(* CoDeSys 2.3.9.50 project: Aerosol_detection_equipment.pro *)
(* Libraries: TcFloatPC.lib 19.10.09 10:19:54, TcUtilities.lib 3.2.16 16:08:58, TcEtherCAT.lib 15.8.22 11:50:34, TcTestAndSet.lib 23.2.09 12:50:08, TcDrive.lib 25.1.17 09:42:28, TcMc2Drive.lib 9.10.17 15:27:28, TcBase.lib 14.5.09 12:14:08, TcSystem.lib 7.6.16 11:01:22, TcBaseMath.lib 27.7.04 12:07:56, TcMath.lib 23.9.04 15:15:30, TcMC2.lib 13.9.17 10:18:38, STANDARD.LIB 5.6.98 12:03:02 *)

(* Task configuration *)
TASK Standard (PRIORITY := 0, INTERVAL := T#10ms);
	MAIN
END_TASK

(* Global variable list: _01_Machine *)
VAR_GLOBAL
(*Signal*)
	stMachine						:ST_Machine;
(*Alarm*)
	arrAlarm							:ARRAY[1..MaxAlarms] OF BOOL;				(*报警号,以Excel为准*)
	arrWarning						:ARRAY[1..MaxAlarms] OF BOOL;				(*提示号,以Excel为准*)

	MSGList1 : ARRAY[1..100] OF BOOL;
	MSGList1_Alarm : BOOL;




(*Info*)
	TaskInfo						:TaskInfoCtrl;
	SysInfo							:SystemInfoCtrl;
	fPlcCycleTime_ms				:LREAL;
(* Global pulse *)
	Pulse							:PulseCtrl;		(*公共脉冲发生器*)
	nPlcTaskCycleTime_ms			:UDINT;			(*PLC周期的毫秒数*)
END_VAR

VAR_GLOBAL CONSTANT
	MaxAlarms			:UINT:=100;
END_VAR

(* Global variable list: _02_System *)
VAR_GLOBAL
	sState						:STRING(20):='MANU';		(*机台当前状态*)
	sStatus						:STRING(20):='INIT'	;			(*当前执行步骤*)

(*系统运行相关指令，面板按钮是输入来源之一*)
	bSysStart					:BOOL;		(*这个start仅指进入自动模式的启动*)
	bSysStop					:BOOL;
	bSysReset					:BOOL;
	bSysEstop					:BOOL;
	bSwitchManualMode			:BOOL;		(*打到了手动模式*)
	bSwitchAutoMode			:BOOL;		(*打到了自动模式*)
	bSysDryRunMode			:BOOL;		(*空跑模式，在触摸屏上选择，不带物料，自动运行的机械检查*)

	bSystemInAutoMode			: BOOL;		(*系统实际处于自动模式*)
	bSystemInManualMode		: BOOL;		(*系统实际处于手动模式*)
	bAutoModeRunning				:BOOL;		(*自动运行中*)

(*系统状态*)
	bGlobalErrorMark				:BOOL;		(*有报警，这个报警时会触发停机的！*)

	bSysStopFlag				:BOOL;		(*停止标记，标记出现，说明进入停机过程*)
	bStopFinished				:BOOL;		(*停止完成*)

(*指令*)
	bResetOnce					:BOOL;		(*单次复位*)
	bhasResetOnce				: BOOL;		(*已经单次复位过了*)
	bForceHomedFlag			:BOOL;		(*强制写回参信号*)
	bBuzzerSilence				:BOOL;		(*消音*)



(*自动状态*)
	eAutoStatus					:EM_Status;		(*自动模式的状态*)

(*机台状态*)
	bAllPowerOnOK				:BOOL;	(*上电检查OK*)
	bDeviceStateOK				:BOOL;	(*总线状态OK*)
	bDriveModeOK				:BOOL;	(*驱动器模式OK*)

	bAutoReady					:BOOL;		(*自动运行的位置条件OK*)
	bAllCylinderBase				:BOOL;		(*所以气缸回到初始位*)

	iSysStatus					:WORD;		(*设备状态*)
	bAirPressureOk:BOOL;(*空气压力是否到位*)



	iActPos_X_Axis					:WORD;						(*	X轴当前位置编码	*)
	iActPos_Z_Axis					:WORD;						(*	Z轴当前位置编码	*)
	iActPos_R_Axis					:WORD;						(*	R轴当前位置编码	*)
	iWarnMoveAbs							:WORD;					(*定位警告信息*)
	iAlarmNetConnect						:WORD;					(*网络连接问题报警信息*)
	iGoHomeTogether_Finish	:	WORD	;	(*一键回原点完成*)
	iGoPrepareAuto_Finish	:	WORD	;	(*一键去准备位完成*)
	iPos_X_Axis				:	WORD	;	(*模组1	X轴目标位置	*)
	iPos_Z_Axis				:	WORD	;	(*模组2	Z轴目标位置	*)
	iPos_X2_Axis				:	WORD	;	(*模组3	X轴目标位置	*)
	iPos_Y2_Axis				:	WORD	;	(*模组4	Y轴目标位置	*)
	iPos_R_Axis				:	WORD	;	(*	R轴目标位置	*)
	iX_Axis_Cmd			:	WORD	;	(*	模组1X轴目标位置运动命令	*)
	iZ_Axis_Cmd			:	WORD	;	(*	模组2Z轴目标位置运动命令	*)
	iX2_Axis_Cmd		:	WORD;		(*	模组3X轴目标位置运动命令	*)
	iY2_Axis_Cmd		:	WORD;		(*	模组4Y轴目标位置运动命令	*)
	iR_Axis_Cmd			:	WORD	;	(*	R轴目标位置运动命令	*)
	iHorizontalAxis_Cmd		:	WORD	;	(*	废物桶检测行程轴目标位置运动命令	*)
	iRotaryAxis_Cmd			:	WORD	;	(*	废物桶检测旋转轴目标位置运动命令	*)
	iLifting_PutPermit_Cmd	:	WORD	;	(*	请求吊装设备放置料筒	*)
	iLifting_GetPermit_Cmd	:	WORD	;	(*	请求吊装设备吊取料筒	*)
	iPos_CollimationAxis		:	WORD	;	(*	准直电机位置	*)
	iCollimationAxis_Cmd	:	WORD	;	(*	准直电机目标位置运动指令	*)
	iRotaryAxisRun_Cmd		:	WORD	;	(*旋转电机一直转*)
	iGoHomeTogether_Cmd	:	WORD	;	(*一键回原点*)
	iGoPrepareAuto_Cmd	:	WORD	;	(*一键去准备位*)
	iGoResetTogether_Cmd	:WORD;		(*一键复位*)
	iGoAutoTogether_Cmd		:WORD;		(*一键启动*)
	iGoStopTogether_Cmd					:WORD;		(*一键停止*)
	iAuto_Cmd				:	WORD	;	(*自动切换*)
	bGoHomeTogether_Cmd	:	BOOL	;	(*一键回原点*)
	bGoPrepareAuto_Cmd	:	BOOL	;	(*一键去准备位*)
	bAuto_Cmd				:	BOOL	;	(*自动切换*)

	bGet_Paper_Cmd:			BOOL;(*取纸*)
	bHasGot_Paper:BOOL;(*取纸完成*)

	bCollect_Cmd:BOOL;(*采集*)
	bHasCollected:BOOL;(*采集完成*)

	bPut_Paper_Cmd:			BOOL;(*放纸*)
	bHasPut_Paper:BOOL;(*放纸完成*)

	bCut_Paper_Cmd:			BOOL;(*裁纸*)
	bHasCut_Paper:BOOL;(*裁纸完成*)

	bSet_Box_Cmd:			BOOL;(*装盒子*)
	bHasSet_Box:BOOL;(*装盒子完成*)



(*报警中间变量*)
	bAxisMovingAbsAlarm			:	ARRAY[1..30] OF BOOL;

(*运行参数*)
	fSetMainVelo_Auto				: 	LREAL;			(*主轴自动速度*)
	fSetMainVelo_Manu				:	LREAL;			(*主轴手动速度*)


(**************************  工艺相关    ****************************************)

(*指令*)
	bEnaleAll						:BOOL;	(*一键使能*)
	bGoHomeTogether				:BOOL;		(*一键回原点*)
	bGoPrepareAuto					:BOOL;		(*一键初始化*)
	bGoResetTogether				:BOOL;		(*一键复位*)
	bGoAutoTogether					:BOOL;		(*一键启动*)
	bGoStopTogether					:BOOL;		(*一键停止*)
	bHeatAll							:BOOL;		(*加热所有*)

(***********************************MODBUS TCP***********************************************)

	mb_Output_Registers : ARRAY[0..255] OF WORD;
	mb_Input_Registers : ARRAY[1..255] OF WORD;

END_VAR

(* Global variable list: _03_Param *)
VAR_GLOBAL CONSTANT
	EIN                             : BOOL  := TRUE;
	AUS                             : BOOL  := FALSE;
	ANZ_SUBSSW                   : UINT   := 5;

	fCurveKp		:REAL:=6.8;		(*角度与毫米的关系*)
END_VAR

VAR_GLOBAL PERSISTENT
	iAxisSoftLimitSwitch_Neg	:ARRAY[1..5] OF BOOL;	(*软限位正限开关*)
	iAxisSoftLimitSwitch_Pos	:ARRAY[1..5] OF BOOL;	(*软限位负限开关*)

	iAxisSoftLimitSwitch_Neg1	:ARRAY[1..5] OF WORD;	(*软限位正限开关*)
	iAxisSoftLimitSwitch_Pos1	:ARRAY[1..5] OF WORD;	(*软限位负限开关*)
	fSaveBias	:ARRAY[1..5] OF REAL;
END_VAR

VAR_GLOBAL

(*运行时数据状态*)
	iAxisSoftLimitSwitch_Neg_Old	:ARRAY[1..5] OF BOOL;	(*软限位正限开关*)
	iAxisSoftLimitSwitch_Pos_Old	:ARRAY[1..5] OF BOOL;	(*软限位负限开关*)
	iMacStateForHmi				:WORD;(*机器状态给HMI*)
END_VAR

(* Global variable list: _04_Motion *)
VAR_GLOBAL
	AxisArr					:ARRAY[1..MaxAxes] OF  axis_ref;		(*PTP轴*)
	Axis_Interface			: ARRAY [1..MAXAxes] OF ST_Axis;		(*轴的PTP控制接口*)
(*功能块定义*)
	aMC_Power				:ARRAY[1..MaxAxes] OF MC_Power;
	aMC_Jog				:ARRAY[1..MaxAxes] OF MC_Jog;
	aMC_Reset				:ARRAY[1..MaxAxes] OF MC_Reset;
	aMC_Halt				:ARRAY[1..MaxAxes] OF MC_Halt;
	aMC_Stop				:ARRAY[1..MaxAxes] OF MC_Stop;
	aMC_SetPos				:ARRAY[1..MaxAxes] OF MC_SetPosition;
	aMC_MoveAbsolute		:ARRAY[1..MaxAxes] OF MC_MoveAbsolute;
	aMC_MoveRelative		:ARRAY[1..MaxAxes] OF MC_MoveRelative;
	aMC_MoveVelocity		:ARRAY[1..MaxAxes] OF MC_MoveVelocity;
	aMC_SetHomeFlag		:ARRAY[1..MaxAxes] OF MC_Home;
	aMC_Home				:ARRAY[1..MaxAxes] OF MC_Home;
	aMC_GearInDyn			:ARRAY[1..MaxAxes] OF MC_GearInDyn;			(*电子齿轮轮耦合*)
	aMC_GearOut			: ARRAY[1..MaxAxes] OF MC_GearOut;		(*电子齿轮轮解耦合*)
	aMC_SoeReset			:ARRAY[1..MaxAxes] OF FB_SoEReset;		(*倍福驱动器复位*)

(*公共状态参数*)
 	Axis_Has_error		:BOOL;		(*任何一根轴有任何错误*)
	Axis_Homing			:BOOL;		(*任何一根轴在回参*)
	All_Enable_OK		:BOOL;		(*所有轴使能成功*)
	All_Homed_OK		:BOOL;		(*所有轴回零成功*)
	bAllAxisAtZero		:BOOL;		(*所有轴都在0位*)
	AllAxesStandStill		:BOOL;		(*所有轴静止*)
(*公共CMD参数*)
	bEnableAll	:	BOOL;	(*使能所有轴*)
(*气缸*)
	stCtrlCylinder	:ARRAY[1..NumOfCylinders]OF ST_Cylinder_Ctrl;
	fbCylinder		:ARRAY[1..NumOfCylinders]OF FB_Cylinder;
END_VAR

VAR_GLOBAL CONSTANT
	MaxAxes							:UINT:=5;		(*轴数，不同于驱动器数，后者是物理轴的个数*)
	NumOfDrives							:UINT:=5;		(*实际驱动器数*)
	MinHomeAxis	:UINT:=1;		(*最小回原点轴*)
	MaxHomeAxis	:UINT:=8;		(*最大回原点轴*)
	NumOfCylinders						:UINT:=38;		(*气缸数*)
END_VAR

(* Global variable list: _05_IO *)
VAR_GLOBAL
	(*数字量输入*)
	El1889s			AT %I*		:ARRAY[1..NumOfDiModule,1..NumOfChannel]OF BOOL;
	(*数字量输出*)
	El2889s 			AT%Q*		:ARRAY[1..NumOfDoModule,1..NumOfChannel]OF BOOL;
	(*模拟量输入*)
	El3064			AT %I*		:ARRAY[1..4]OF INT;
	(*实际驱动器作为EtherCAT伺服的个数  ETHERCAT状态*)
	DrivesOP 		AT %I*		:ARRAY[1..NumOfDrives]OF UINT;
	(*驱动器的模式输出，8为位置模式*)
	iSetDriveMode 	AT %Q*		:ARRAY [1..NumOfDrives] OF SINT := NumOfDrives(CSP);
	(*驱动器返回的控制模式*)
	iActDriveMode	AT%I*		:ARRAY[1..NumOfDrives]OF SINT;
	(*驱动器上的IO监控，EL2521不包含*)
	iDriveDI			AT%I*  :ARRAY [1..NumOfDrives] OF INT;
	(*驱动器上的电流监控，EL2521不包含*)
	iMotorTorque		 AT%I*  :ARRAY [1..NumOfDrives] OF INT;

END_VAR


VAR_GLOBAL CONSTANT
	NumOfDiModule		:UINT:=7;		(*DI输入模块总数*)
	NumOfDoModule		:UINT:=3;		(*DO输出模块总数*)
	NumOfAiModule		:UINT:=0;		(*DI输入模块总数*)
	NumOfChannel		:UINT:=16;		(*IO模块的通道数*)

	iEcatOp				:UINT:=8;
	CSP					:USINT:=8;
	CSV					:USINT:=9;
	CST					:USINT:=10;
END_VAR

(* Global variable list: _06_Hmi *)
VAR_GLOBAL
(***********************HMI变量****************************)
(********  指令 ***********)
	stHmiCmd			:	ST_HmiCmd;
	stHmiAxisCmd			:	ARRAY[1..MaxAxes] OF ST_AxisCmd;
(********  显示 ***********)
	stHmiDisplay				:	ST_HmiDisplay;
	stAxisDisplay			:	ARRAY[1..MaxAxes] OF ST_AxisDisplay;
END_VAR


VAR_GLOBAL PERSISTENT
(********  参数 ***********)
	stAxisParam			:	ARRAY[1..MaxAxes] OF ST_AxisParam;
END_VAR

(* Global variable list: TwinCAT_Configuration *)
(* Generated automatically by TwinCAT - (read only) *)
VAR_CONFIG
	.AxisArr[1].PlcToNc AT %QB53 : PLCTONC_AXIS_REF;	(*  ~ {LinkedWith:TINC^NC-Task 1 SAF^Axes^Axis 1^Inputs^Axis 1_FromPlc} *)
	.AxisArr[1].NcToPlc AT %IB155 : NCTOPLC_AXIS_REF;	(*  ~ {LinkedWith:TINC^NC-Task 1 SAF^Axes^Axis 1^Outputs^Axis 1_ToPlc} *)
	.AxisArr[2].PlcToNc AT %QB181 : PLCTONC_AXIS_REF;	(*  ~ {LinkedWith:TINC^NC-Task 1 SAF^Axes^Axis 2^Inputs^Axis 2_FromPlc} *)
	.AxisArr[2].NcToPlc AT %IB283 : NCTOPLC_AXIS_REF;	(*  ~ {LinkedWith:TINC^NC-Task 1 SAF^Axes^Axis 2^Outputs^Axis 2_ToPlc} *)
	.AxisArr[3].PlcToNc AT %QB309 : PLCTONC_AXIS_REF;	(*  ~ {LinkedWith:TINC^NC-Task 1 SAF^Axes^Axis 3^Inputs^Axis 3_FromPlc} *)
	.AxisArr[3].NcToPlc AT %IB411 : NCTOPLC_AXIS_REF;	(*  ~ {LinkedWith:TINC^NC-Task 1 SAF^Axes^Axis 3^Outputs^Axis 3_ToPlc} *)
	.AxisArr[4].PlcToNc AT %QB437 : PLCTONC_AXIS_REF;	(*  ~ {LinkedWith:TINC^NC-Task 1 SAF^Axes^Axis 4^Inputs^Axis 4_FromPlc} *)
	.AxisArr[4].NcToPlc AT %IB539 : NCTOPLC_AXIS_REF;	(*  ~ {LinkedWith:TINC^NC-Task 1 SAF^Axes^Axis 4^Outputs^Axis 4_ToPlc} *)
	.AxisArr[5].PlcToNc AT %QB565 : PLCTONC_AXIS_REF;	(*  ~ {LinkedWith:TINC^NC-Task 1 SAF^Axes^Axis 5^Inputs^Axis 5_FromPlc} *)
	.AxisArr[5].NcToPlc AT %IB667 : NCTOPLC_AXIS_REF;	(*  ~ {LinkedWith:TINC^NC-Task 1 SAF^Axes^Axis 5^Outputs^Axis 5_ToPlc} *)
	.El1889s AT %IB0 : ARRAY [1..7, 1..16] OF BOOL;
	.El2889s AT %QB0 : ARRAY [1..3, 1..16] OF BOOL;
	.El3064 AT %IB112 : ARRAY [1..4] OF INT;
	.DrivesOP AT %IB120 : ARRAY [1..5] OF UINT;
	.iSetDriveMode AT %QB48 : ARRAY [1..5] OF SINT;
	.iActDriveMode AT %IB130 : ARRAY [1..5] OF SINT;
	.iDriveDI AT %IB135 : ARRAY [1..5] OF INT;
	.iMotorTorque AT %IB145 : ARRAY [1..5] OF INT;
END_VAR

(* Data type in 01_States *)
TYPE EM_State :	(*机台或者部件的几种状态*)
(
	PowerOn,
	ConnectionTest,
	Init,
	Manu,
	Auto,
	Error
);
END_TYPE

(* Data type in 01_States *)
TYPE EM_Status :	(*自动模式下的几个流程*)
(
	AUTO_STOP       :=   0,
	AUTO_W_RUN      :=   2,
	AUTO_RUN        :=   3,
	AUTO_W_HALT     :=   4,
	AUTO_HALT       :=   5,
	AUTO_W_STOP     :=   6
);
END_TYPE

(* Data type in 04_AxisControl *)
TYPE ST_Axis :	(*Johnson made this on 2017-01-17*)
STRUCT
(*status*)
	AxisName		:STRING(31);		(*轴名称*)
	AxisID			:UDINT;		(*轴在NC中的编号*)

	Axis_Limit_Neg	:BOOL;		(*负限位触发信号*)
	Axis_Limit_Pos	:BOOL;		(*正限位触发信号*)
	Axis_HomeSwitch	:BOOL;		(*原点触发信号*)
	Axis_Ready		:BOOL;
	Axis_Err			:BOOL;
	Axis_ErrID		:UDINT;

	Axis_Homed		:BOOL;
	Axis_Homing		:BOOL;
	Axis_Coupled		:BOOL;
	Axis_NotMoving	:BOOL;

	fActPos			:LREAL;
	fActPosModbus			:WORD;
	fActVelo			:LREAL;
	fScaleFactor		:LREAL;
(*Command*)
	bEnable			:BOOL;		(*使能*)
	bEnableFw		:BOOL:=TRUE;		(*正向使能*)
	bEnableBw		:BOOL:=TRUE;		(*负向使能*)
	bJog_Fw			:BOOL;		(*正向点动*)
	bJog_Bw		:BOOL;		(*反向点动*)

	bHalt			:BOOL;	(*暂停*)
	bStop			:BOOL;	(*停止*)
	bReset			:BOOL;	(*复位*)

	bMoveAbs		:BOOL;	(*运行绝对位置*)
	bMoveRel		:BOOL;	(*运行当对位置*)
	bMoveVelo		:BOOL;	(*向一个方向持续运行，方向由前面的正向点动或者反向点动设置*)

	bHome			:BOOL;		(*启动回参*)
	bSetPos			:BOOL;		(*设置轴当前的位置为一个绝对位置*)

	bCamIn			:BOOL;
	bCamOut		:BOOL;

	bGearIn			:BOOL:=FALSE;
	bGearOut		:BOOL:=FALSE;

	fGearInDynAcc	:LREAL:=50000;
	fGearInDynDec	:LREAL:=50000;
	fGearRatio		:LREAL;		(*电子齿轮耦合齿轮比*)

	nCmdMode		:SINT;(*8=CSP位置, 9=CSV,10=CST力矩*)
(*Parameter*)
	fOverride			 :LREAL:=100;		(*MC_power中实际倍率的设定，默认值为100*)
	fPositon_of_Abs	 :LREAL;		(*绝对位置位移*)
	fPosition_of_Rel	 :LREAL;		(*相对位置位移*)
	fVelocity_of_Abs	 :LREAL:=5;		(*位置移动速度，包含相对位移和绝对位移指令的速度*)
	fVelocity_of_Rel	 :LREAL;		(*位置移动速度，包含相对位移和绝对位移指令的速度*)
	fVelocity_of_Velo	 :LREAL;		(*速度指令下的运动速度，用在mc_movevelocity里面*)
	fVelocity_of_Jog	 :LREAL:=5;		(*手动点动速度，可以在程序里面设置不同值*)

	fAcc				:LREAL:=0;(*0代表使用SystemManager里面的参数*)
	fDec			:LREAL:=0;
	fJerk			:LREAL:=0;
	fPosition_ToBeSet	:LREAL;		(*setpos功能块将轴当前的位置设置为这个变量*)
	fRefPos				:LREAL:=0;		(*使用TwinCAT PLC的MC_Home回零时，将外部信号设成这个值*)

	bInVelo			:BOOL;		(*速度模式，达到了速度*)
END_STRUCT
END_TYPE

(* Data type in 05_Function/02_Axis *)
TYPE ST_AxisCmd :
STRUCT
(*Command*)
	bEnable				:BOOL(*:=TRUE*);
	bJog_Fw			:BOOL;		(*正向点动*)
	bJog_Bw			:BOOL;		(*反向点动*)
	bJog_InchingFw			:BOOL;		(*正向寸动*)
	bJog_InchingBw			:BOOL;		(*反向寸动*)
	bMoveToZero				:BOOL;		(*回原点*)		(*正负极直线电机回原点，纠偏和切刀回原点，短路测试电机回原点，叠台...*)
	bMoveAbs				:BOOL;
	bMoveRel				:BOOL;
	bReset					:BOOL;
	bHome					:BOOL;
	bSetPos					:BOOL;
	bSetBiasBnt			:BOOL;		(*保存原点按钮*)
END_STRUCT
END_TYPE

(* Data type in 05_Function/02_Axis *)
TYPE ST_AxisDisplay :
STRUCT
(*DisPlay*)
	bError			:BOOL;		(*报错*)
	bEnabled		:BOOL;		(*使能*)
	bHoming			:BOOL;		(*回参中*)
	bHomed			:BOOL;		(*回参完成*)
	bMoiving		:BOOL;		(*移动中*)
	bPosLimit		:BOOL;
	bNegLimit		:BOOL;
	udiErrorId		:UDINT;		(*轴错误代码*)

	fActPos	 		:REAL:=15;			(*轴当前位置*)
(*	fActModPos		:REAL:=0;	*)
	fActVelo		:REAL:=5;			(*轴当前速度*)
	fOverride		:REAL:=100;			(*轴当前速比值*)

END_STRUCT
END_TYPE

(* Data type in 05_Function/02_Axis *)
TYPE ST_AxisParam :
STRUCT
(*Parameter，头两个参数可以用触摸屏上设置*)
	fVelocity_of_Jog	 		:LREAL:=4;			(*手动点动速度，可以在程序里面设置不同值*)
	fInchingDistance			:LREAL:=1;			(*寸动距离，可以在程序里面设置不同值*)
	fVelo_of_Posi			:REAL:=15;		(*手动定位速度*)

	fVelo_of_Auto		:LREAL:=6;		(*自动速度*)
	fVelocity_of_Abs		:LREAL:=6;
	fTargetPos				:LREAL;

	fOverride				:LREAL:=100;			(*实际倍率的设定，默认值为100*)
	SavedPosition			:LREAL:=0;
	iTargetNr				:UINT;
	ZeroPos				:REAL;		(*零位，原点开关决定*)
	StandbyPos			:REAL;		(*待机位*)
	WorkPos1			:REAL;		(*工位1*)
	WorkPos2			:REAL;		(*工位2*)
	WorkPos3			:REAL;		(*工位3*)

	fTargetPosi			:REAL;		(*目标定位*)
END_STRUCT
END_TYPE

(* Data type in 04_AxisControl *)
TYPE ST_Cylinder_Ctrl :	(*Johnson made this on 2017-01-17*)
STRUCT
(*From DI*)
	DiBaseLimit				:BOOL;		(*负限位触发信号*)
	DiWorkLimit				:BOOL;		(*正限位触发信号*)

(*To Do*)
	DoAct			:BOOL;		(*动作*)
	DoBack			:BOOL;		(*回到base位*)

(*To PLC status*)
	CylinderName		:STRING(31);		(*气缸名称*)
	CylinderID			:UDINT;				(*气缸编号*)

	Cylinder_Limit_Base	:BOOL;		(*负限位触发信号*)
	Cylinder_Limit_Work	:BOOL;		(*正限位触发信号*)
	CylinderAlarm_TimeOut	:BOOL;			(*气缸动作超时*)

(*PLC commmand*)
	bAct			:BOOL;		(*动作*)
	bBack			:BOOL;		(*回到base位*)
	bSwitch			:BOOL;		(*切换*)


(*Parameter*)
	bContinue				:BOOL;	(*是否连续运动气缸*)
	fTimeOfContinue			:REAL:=1;
	fTimeOfOvertime			:REAL:=1;		(*单位秒*)

END_STRUCT
END_TYPE

(* Data type in 05_Function/01_Machine *)
TYPE ST_HmiCmd :
STRUCT

(***************************************************   系统    ********************************************)

	bStart		:BOOL;
	bStop		:BOOL;
	bReset		: BOOL;		(*HMI上的复位*)
	bEstop		: BOOL;		(*HMI上的急停*)
	bNtReboot		: BOOL;		(*系统重启*)
	bNtShutdown	: BOOL;		(*系统关机*)
	bSaveData		: BOOL;		(*保存系统设置参数*)
	bSilence			: BOOL;		(*消音按钮*)
END_STRUCT
END_TYPE

(* Data type in 05_Function/01_Machine *)
TYPE ST_HmiDisplay :
STRUCT

(***************************************************  设备状态     ********************************************)

	bAll_Enable_OK				:BOOL;	(*所有轴使能成功*)
	bAll_Homed_OK				:BOOL;	(*所有轴回零成功*)
	bAutoReady					:BOOL;	(*运行准备信号，满足了打到自动的准备条件*)
	bAutoSwitch				:BOOL;	(*在界面上显示当前旋转开关处于手动还是自动,True为自动，false为手动*)
	bAutoMode					:BOOL;	(*设备进入了自动模式*)
	bAutoRunning  				:BOOL;	(*自动运行中*)
	bHeartBeat					:BOOL;
	iMachineState			:		UINT;		(*机台状态*)
(***************************************************  系统     ********************************************)
	sProgram_Vision				:STRING;	(*程序版本号*)


END_STRUCT
END_TYPE

(* Data type in 03_Machine *)
TYPE ST_Machine :
STRUCT

(***************************************************   DI    ********************************************)
	btnStart			:BOOL;	(*	启动按钮	*)
	btnStop			:BOOL;	(*	停止按钮	*)
	btnReset		:BOOL;	(*	复位按钮	*)
	bswAutoSwitch	:BOOL;	(*	手自动切换按钮	*)
	btnEstop		:BOOL;	(*	急停按钮	*)
	bSingle			:BOOL;



(***************************************************   DO    ********************************************)

	boLamp_Red		:BOOL;	(*	灯柱-红	*)
	boLamp_Green	:BOOL;	(*	灯柱-绿	*)
	boLamp_Yellow	:BOOL;	(*	灯柱-黄	*)
	boBuzzer		:BOOL;	(*	蜂鸣器	*)
	boBtnStartLed	:BOOL;	(*启动按钮指示灯，绿色*)
	boBtnStopLed	:BOOL;	(*停止按钮指示灯，红色*)
	boBtnResetLed	:BOOL;	(*复位按钮指示灯，橙色*)
END_STRUCT
END_TYPE

(* POU MAIN, ST *)
PROGRAM MAIN
VAR
	MainState					:EM_State;	(*主程序步，其他程序可以读*)
	bFirstCycle: BOOL:=TRUE;	(*初始化用的*)
(*保存掉电保持参数*)
	FB_WritePersistentData1: FB_WritePersistentData;
	tCycleTimer:TON;
	bWrite: BOOL;

(*系统重启*)
	tNtDelayReset:TON;
	bReboot: BOOL;	(*重启系统的变量*)
	NT_Reboot1: NT_Reboot;

(*系统关机*)
	NT_Shutdown1: NT_Shutdown;
	tNtDelayShutdown: TON;
	bShutdown: BOOL;

(*远程桌面接管*)
	OpenRemoteDesktop: NT_StartProcess;
	timerHMI	:TON;

(*设置系统时间*)
	TimeToBeSet: TIMESTRUCT;
	bSetTime: BOOL;
	NT_SetLocalTime_1: NT_SetLocalTime;
(*系统时间获取*)
	NT_GetTime1: NT_GetTime;
	GetTimeStartDelay:TON;
	TIMESTR1				:TIMESTRUCT;

	i: UINT;

(*
(*计算加工时间相关变量*)
	j:UINT;(*表格的FOR序号*)
	n:UINT:=1;
	rtrigAutoRunning:R_TRIG;	(*自动运行上升沿*)
	ftrigAutoRunning:F_TRIG;	(*自动运行下升沿*)
	nStopLock: BOOL;
	itets: UINT;
(*其它*)
	R_TRIG_Enabled: R_TRIG;
	BalanceLumpDeclineDelay:TON;(*配重块下降到下限传感器位置后延时一定时间才停止*)
	nParameterUpdateTop:BOOL;(*参数被更改，提醒用户更新运行数据*)
	ActTableModeNumber: BOOL;	(*表格序号至少一个被激活*)
*)
	rtrigStart,rtrigReset,rtrigStop: R_TRIG;
	fTrigAutoManulMode: F_TRIG;
	rTrigAutoManualMode: R_TRIG;
	tDelayManualMode:TON;(*打到手动的延时*)
(*Lamp and Buzzer*)
	eStepBuzze: UINT;
	rTrigBuzze: R_TRIG;
	tDelayBuzze: TON;



	LagDistance_ZM: LREAL;
	LagDistance_CM: LREAL;
	FirstCycle_Step: UINT;
	R_TRIGbDriveModeOK:R_TRIG;
	tDelay:TON;
END_VAR
PRG_IO.Input();
PRG_Alarm();
PRG_Monitor();
PRG_Auto.Act_Modbus_TCP();
MAIN._NT;
MAIN.Command;
MAIN.Status;

CASE MainState OF
PowerOn:
	PRG_Power();
	MainState:=ConnectionTest;

ConnectionTest:
	IF bDeviceStateOK AND bDriveModeOK  THEN
		bResetOnce:=TRUE;
		MainState:=INIT;
		PRG_ServOn();
	END_IF

INIT:	(*程序的初始化处理，并非机器的工艺初始化*)
	PRG_Init();
	IF All_Enable_OK OR bHasResetOnce   THEN
		MainState:=MANU;
	ELSIF Axis_Has_error THEN
		MainState:=ConnectionTest;		(*轴有错就再复位一次,这个时针对有的驱动在PLC之前启动好，PLC连接时会报通讯错误，需要复位一次*)
		bHasResetOnce:=TRUE;
	END_IF

MANU:
(*手动模式*)
	PRG_Manual;
	IF bSysEstop  THEN			(*急停也是从手动中进入的*)
		MainState:=ERROR;
	ELSIF
		bSwitchAutoMode
		AND NOT bGlobalErrorMark
		AND NOT bSysEstop
		AND bAutoReady
	THEN
		MainState:=AUTO;
	END_IF

AUTO:
	PRG_Auto();
	IF  bSysEstop (*AND bStopFinished*) THEN	(*急停触发，并且停好了*)
		MainState:=ERROR;
	ELSIF bSwitchManualMode AND NOT bStopFinished THEN
		MainState:=MANU;
	END_IF
ERROR:
	PRG_Estop();
	IF NOT bSysEstop THEN
		MainState:=PowerOn;
		bResetOnce:=TRUE;
	END_IF
END_CASE


IF( bSysEstop AND MainState<>AUTO) (*OR bGlobalErrorMark *)THEN		(*非自动模式下的急停处理*)
	MainState:=ERROR;
END_IF
PRG_M_Function();
PRG_PTP();
PRG_Auto.Act_Run();
PRG_IO.Output();
END_PROGRAM
ACTION _NT:
(*系统重启，CE远程桌面，系统时间，定时保存掉电数据，等系统常规动作*)

tNtDelayReset(IN:=bReboot , PT:=t#3s , Q=> , ET=> );
NT_Reboot1(
	NETID:='' ,
	DELAY:= ,
	START:=(*tNtDelayReset.Q  ,*),
	TMOUT:=DEFAULT_ADS_TIMEOUT ,
	BUSY=> ,
	ERR=> ,
	ERRID=> );

tNtDelayShutdown(IN:=bShutdown , PT:=t#0.5s , Q=> , ET=> );
NT_Shutdown1(
	NETID:= ,
	DELAY:= ,
	START:=tNtDelayShutdown.Q,			(*针对win7系统用的，CE系统直接断电*)
	TMOUT:=DEFAULT_ADS_TIMEOUT ,
	BUSY=> ,
	ERR=> ,
	ERRID=> );

(******************* 开启CE系统远程桌面  ******************************************)
timerHMI(IN:=bFirstCycle, PT:=T#2S);
(*IF timerHMI.Q THEN
	bFirstCycle:=FALSE;
END_IF*)
OpenRemoteDesktop(
	NETID:='' ,
	PATHSTR:='\windows\CerDisp.exe' ,
	DIRNAME:='\windows' ,
	COMNDLINE:= ,
	START:=(*timerHMI.Q*) ,		(*建议第一次通过程序手动开启远程桌面之后，再修改注册表种launch90的值，以及增加Enable远程的注册表文件到regfile中来实现*)
	TMOUT:= ,
	BUSY=> ,
	ERR=> ,
	ERRID=> );
(********************** 获取系统时间   ***************************************)


GetTimeStartDelay(IN:=NOT GetTimeStartDelay.Q  , PT:=T#2s , Q=> , ET=> );
NT_GetTime1(
	NETID:= ,
	START:=GetTimeStartDelay.Q ,
	TMOUT:= , 
	BUSY=> ,
	ERR=> ,
	ERRID=> ,
	TIMESTR=>TIMESTR1 );

TIMESTR1.wYear;		(*年*)
TIMESTR1.wMonth;		(*月*)
TIMESTR1.wDay;		(*日*)
TIMESTR1.wHour;		(*时*)
TIMESTR1.wMinute;		(*分*)
TIMESTR1.wSecond;		(*秒*)
TIMESTR1.wMilliseconds;	(*毫秒*)
TIMESTR1.wDayOfWeek;	(*星期*)

(********************** 设置系统时间   ***************************************)
NT_SetLocalTime_1(
	NETID:= , 
	TIMESTR:=TimeToBeSet ,
	START:=bSetTime ,
	TMOUT:=t#500ms ,
	BUSY=> , 
	ERR=> ,
	ERRID=> );
TimeToBeSet.wYear;			(*年*)
TimeToBeSet.wMonth;		(*月*)
TimeToBeSet.wDay;			(*日*)
TimeToBeSet.wHour;			(*时*)
TimeToBeSet.wMinute;		(*分*)
TimeToBeSet.wSecond;		(*秒*)
TimeToBeSet.wMilliseconds;	(*毫秒*)
TimeToBeSet.wDayOfWeek;	(*星期*)

(***********************  保存掉电保持数据   **************************************)
tCycleTimer(IN:=NOT tCycleTimer.Q , PT:=t#60s , Q=>bWrite , ET=> );
FB_WritePersistentData1(
	NETID:='' ,
	PORT:=801 ,
	START:=bWrite OR stHmiCmd.bSaveData OR SystemtaskInfoArr[1].firstCycle  ,
	TMOUT:=t#500ms ,
	MODE:=SPDM_2PASS ,
	BUSY=> ,
	ERR=> ,
	ERRID=> );
(**********************  系统周期时间获取   ***************************************)
nPlcTaskCycleTime_ms:=SystemtaskInfoArr[1].cycleTime/10000;


(******************* 伺服位置设置********************)
R_TRIGbDriveModeOK(CLK:=(bDriveModeOK), Q=> );
IF (R_TRIGbDriveModeOK.Q AND timerHMI.Q) OR (FirstCycle_Step=0 AND MainState=MANU)  THEN
		FirstCycle_Step:=100;
END_IF



tDelay(IN:= , PT:=t#20ms , Q=> , ET=> );

CASE FirstCycle_Step OF
0:
;
100:
	tDelay.IN:=TRUE;
	IF tDelay.Q THEN
		FirstCycle_Step:=110;
	END_IF
110:
	tDelay.IN:=FALSE;
	FOR i:=1 TO 5 DO
		Axis_Interface[i].fPosition_ToBeSet := -fSaveBias[i]+AxisArr[i].NcToPlc.ActPos;
	END_FOR
	FirstCycle_Step:=200;
200:
	FOR i:=1 TO 5 DO
		Axis_Interface[i].bSetPos:=TRUE;(*触发信号*);
	END_FOR
	FirstCycle_Step:=300;
300:
	bFirstCycle:=FALSE;
	FirstCycle_Step:=400;
400:
	;
END_CASE
END_ACTION
ACTION Command:
(*系统状态切换按钮的响应与信号汇总，以及指示灯的输出*)

rtrigStart(CLK:=stMachine.	btnStart OR stHmiCmd.bStart , Q=> );		(*如果有其他HMI触发的信号也写到此处*)
rtrigStop(CLK:=stMachine.	btnStop OR stHmiCmd.bStop, Q=> );
rtrigReset(CLK:=stMachine.	btnReset OR stHmiCmd.bReset OR bResetOnce, Q=> );

tDelayManualMode(IN:=NOT (stMachine.bswAutoSwitch OR bAuto_Cmd),PT:=t#1s,Q=>,ET=>);(*下降沿延迟*)
rTrigAutoManualMode(CLK:=stMachine.bswAutoSwitch OR bAuto_Cmd, Q=> );		(*打到自动的上升沿*)
fTrigAutoManulMode(CLK:=tDelayManualMode.Q, Q=> );		(*下降沿信号*)


IF bResetOnce THEN
	bResetOnce:=FALSE;		(*触发后将信号复位掉*)
END_IF

(*模式选择*)
IF  rTrigAutoManualMode.Q THEN
	bSwitchAutoMode:=TRUE;
	bSwitchManualMode:=FALSE;
ELSIF tDelayManualMode.Q AND NOT stMachine.bswAutoSwitch  THEN
	bSwitchAutoMode:=FALSE;
	bSwitchManualMode:=TRUE;
END_IF

(*自动运行判定*)
bAutoModeRunning;
bSystemInManualMode:=(MainState=MANU);
bSystemInAutoMode:=(MainState=AUTO);


(*单次触发的信号*)
bSysStart:=rtrigStart.Q ;
bSysStop:=rtrigStop.Q;
bSysReset:=rtrigReset.Q ;
bSysEstop:=stMachine.btnEstop;




bBuzzerSilence:=stHmiCmd.bSilence;	(*触摸屏选择消音,彻底不报警*)




(********************************** Systemfunctions **********************************************************)
	SysInfo(
		Reset				:= ,
		TimeStampTrig		:= Pulse._100ms.RT,
		RunTimeNo			=> ,
		ProjectName			=> ,
		NumberOfTasks		=> ,
		OnlineChangeCount	=> ,
		RetainVarErr		=> ,
		PersistenVarErr		=> ,
		TimeStampDT			=> ,
		TimeStamp			=> ,
		TimeStr				=> ,
		DateStr				=> ,
		TimeStamp2			=> ,
		TimeStruct			=> ,
		MonthDays			=> ,
		LeapYear			=> ,
		WeekOfYear			=> ,
		timezoneId			=>);

	TaskInfo(
		index				=> ,
		active				=> ,
		taskName			=> ,
		firstCycle			=> ,
		cycleTimeExceeded	=> ,
		cycleTime			=> ,
		lastExecTime		=> ,
		priority			=> ,
		cycleCount			=> );

	Pulse(
		BlinkSlow			=> ,
		Blink				=> ,
		BlinkFast			=> );
END_ACTION
ACTION Status:
(*系统灯*)

CASE eStepBuzze OF
	0:
	(*系统故障或者急停时*)
		rTrigBuzze(CLK:=bGlobalErrorMark OR bSysEstop  , Q=> );
		IF rTrigBuzze.Q
		THEN
			eStepBuzze:=10;
			tDelayBuzze(IN:= TRUE, PT:=t#3s , Q=> , ET=> );
		END_IF
	10:
		stMachine.boBuzzer:=bGlobalErrorMark AND Pulse._1s.Q;
		tDelayBuzze(IN:= TRUE, PT:=t#3s , Q=> , ET=> );
		IF tDelayBuzze.Q
		THEN
			eStepBuzze:=0;
			tDelayBuzze(IN:= FALSE, PT:=t#3s , Q=> , ET=> );
			stMachine.boBuzzer:=FALSE;
		END_IF
END_CASE


IF bGlobalErrorMark
THEN										(*报错，红灯*)
	stMachine.boLamp_Green:=FALSE;
	stMachine.boLamp_Red:=TRUE;
	stMachine.boLamp_Yellow:=FALSE;

	stMachine.boBtnStopLed:=TRUE;
	stMachine.boBtnStartLed:=FALSE;
	stMachine.boBtnResetLed:=FALSE;
ELSIF MainState=AUTO (*AND bAutoModeRunning*)					(*自动模式，并且运动起来了*)
THEN
	stMachine.boLamp_Green:=bAutoModeRunning;
	stMachine.boLamp_Red:=FALSE;
	stMachine.boLamp_Yellow:=FALSE;

	stMachine.boBtnStopLed:=FALSE;
	stMachine.boBtnStartLed:=TRUE;
	stMachine.boBtnResetLed:=FALSE;
ELSE										(*手动，黄灯*)
	stMachine.boLamp_Green:=FALSE;
	stMachine.boLamp_Red:=FALSE;
	stMachine.boLamp_Yellow:=TRUE;

	stMachine.boBtnStopLed:=FALSE;
	stMachine.boBtnStartLed:=FALSE;
	stMachine.boBtnResetLed:=TRUE;
END_IF


CASE MainState OF
PowerOn:			stHmiDisplay.iMachineState:=0;
ConnectionTest:		stHmiDisplay.iMachineState:=1;
MANU:			stHmiDisplay.iMachineState:=2;iSysStatus:=1;
AUTO:
	IF NOT bAutoModeRunning THEN stHmiDisplay.iMachineState:=3;
	ELSE	stHmiDisplay.iMachineState:=4;iSysStatus:=2;
	END_IF

ERROR:	stHmiDisplay.iMachineState:=5;iSysStatus:=3;
END_CASE

stHmiDisplay.bHeartBeat:=Pulse._1s.Q;
END_ACTION

(* POU 01_IO/PRG_IO, ST *)
PROGRAM PRG_IO
VAR
	Filter:ARRAY[1..20]OF TON;		(*信号滤波*)

	MINLeftAngleValue: REAL;
	MaxLeftAngleValue: REAL;
	bfirst: BOOL := TRUE;
	fError: REAL;

	fAiFilterKp:REAL:=0.8;
	I: INT;

	iVoltage:REAL;
	fbAiFilter:Aifilter;
END_VAR
;
END_PROGRAM
ACTION Input:
(***************************** DI1   ********************************************)
stMachine.	btnStart	:=	El1889s[1,1]	;	(*启动按钮*)
stMachine.	btnStop	:= 	El1889s[1,2]	;	(*停止按钮*)
stMachine.	btnReset	:=	El1889s[1,3]	;	(*复位按钮*)
stMachine.	btnEstop	:=	Filter[1].Q;	(*急停按钮*)
Filter[1](IN:=NOT El1889s[1,4] , PT:=t#500ms , Q=> , ET=> );(*防止开机触发*)
bAirPressureOk:= El1889s[1,5]; (*空气压力到位*)


(***************************** DI2   ********************************************)
stCtrlCylinder[1].DiBaseLimit	:=El1889s[2,1];	(*采集盖下压气缸1基始位*)
stCtrlCylinder[1].DiWorkLimit	:=El1889s[2,2];	(*采集盖下压气缸1工作位*)
stCtrlCylinder[2].DiBaseLimit	:=El1889s[2,3];	(*采集盖下压气缸2基始位*)
stCtrlCylinder[2].DiWorkLimit	:=El1889s[2,4];	(*采集盖下压气缸2工作位*)
stCtrlCylinder[3].DiBaseLimit	:=El1889s[2,5];	(*滤纸转运组吸盘气缸基始位*)
stCtrlCylinder[3].DiWorkLimit	:=El1889s[2,6];	(*滤纸转运组吸盘气缸工作位*)
stCtrlCylinder[4].DiBaseLimit	:=El1889s[2,7];	(*气动拧瓶盖组瓶盖夹爪气缸基始位*)
stCtrlCylinder[4].DiWorkLimit	:=El1889s[2,8];	(*气动拧瓶盖组瓶盖夹爪气缸工作位*)
stCtrlCylinder[5].DiBaseLimit	:=El1889s[2,9];	(*气动拧瓶盖组?升降动作气缸基始位*)
stCtrlCylinder[5].DiWorkLimit	:=El1889s[2,10];	(*气动拧瓶盖组?升降动作气缸工作位*)
stCtrlCylinder[6].DiBaseLimit	:=El1889s[2,11];	(*气动拧瓶盖组 ?水平动作?气缸基始位*)
stCtrlCylinder[6].DiWorkLimit	:=El1889s[2,12];	(*气动拧瓶盖组 ?水平动作?气缸工作位*)
stCtrlCylinder[7].DiBaseLimit	:=El1889s[2,13];	(*装盒子组?料盒切换动作气缸基始位*)
stCtrlCylinder[7].DiWorkLimit	:=El1889s[2,14];	(*装盒子组?料盒切换动作气缸工作位*)
stCtrlCylinder[8].DiBaseLimit	:=El1889s[2,15];	(*装盒子组?定位夹紧气缸1基始位*)
stCtrlCylinder[8].DiWorkLimit	:=El1889s[2,16];	(*装盒子组?定位夹紧气缸1工作位*)

(***************************** DI3   ********************************************)

stCtrlCylinder[9].DiBaseLimit	:=el1889s[3,1];	(*装盒子组?定位夹紧气缸2基始位*)
stCtrlCylinder[9].DiWorkLimit	:=el1889s[3,2];	(*装盒子组?定位夹紧气缸2工作位*)
stCtrlCylinder[10].DiBaseLimit	:=el1889s[3,3];	(*装盒子组?戳纸升降气缸基始位*)
stCtrlCylinder[10].DiWorkLimit	:=el1889s[3,4];	(*装盒子组?戳纸升降气缸工作位*)
stCtrlCylinder[11].DiBaseLimit	:=el1889s[3,5];	(*裁剪组?压板升降气缸基始位*)
stCtrlCylinder[11].DiWorkLimit	:=el1889s[3,6];	(*裁剪组?压板升降气缸工作位*)
stCtrlCylinder[12].DiBaseLimit	:=el1889s[3,7];	(*裁剪组?裁剪冲压气缸基始位*)
stCtrlCylinder[12].DiWorkLimit	:=el1889s[3,8];	(*裁剪组?裁剪冲压气缸工作位*)
stCtrlCylinder[13].DiBaseLimit	:=el1889s[3,9];	(*裁剪组?防漏气缸基始位*)
stCtrlCylinder[13].DiWorkLimit	:=el1889s[3,10];	(*裁剪组?防漏气缸工作位*)
stCtrlCylinder[14].DiBaseLimit	:=el1889s[3,11];	(*裁剪组?单戳纸气缸1基始位*)
stCtrlCylinder[14].DiWorkLimit	:=el1889s[3,12];	(*裁剪组?单戳纸气缸1工作位*)
stCtrlCylinder[15].DiBaseLimit	:=el1889s[3,13];	(*裁剪组?单戳纸气缸2基始位*)
stCtrlCylinder[15].DiWorkLimit	:=el1889s[3,14];	(*裁剪组?单戳纸气缸2工作位*)
stCtrlCylinder[16].DiBaseLimit	:=el1889s[3,15];	(*裁剪组?单戳纸气缸3基始位*)
stCtrlCylinder[16].DiWorkLimit	:=el1889s[3,16];	(*裁剪组?单戳纸气缸3工作位*)

(***************************** DI4   ********************************************)

stCtrlCylinder[17].DiBaseLimit	:=el1889s[4,1];	(*裁剪组?单戳纸气缸4基始位*)
stCtrlCylinder[17].DiWorkLimit	:=el1889s[4,2];	(*裁剪组?单戳纸气缸4工作位*)
stCtrlCylinder[18].DiBaseLimit	:=el1889s[4,3];	(*裁剪组?单戳纸气缸5基始位*)
stCtrlCylinder[18].DiWorkLimit	:=el1889s[4,4];	(*裁剪组?单戳纸气缸5工作位*)
stCtrlCylinder[19].DiBaseLimit	:=el1889s[4,5];	(*裁剪组?单戳纸气缸6基始位*)
stCtrlCylinder[19].DiWorkLimit	:=el1889s[4,6];	(*裁剪组?单戳纸气缸6工作位*)
stCtrlCylinder[20].DiBaseLimit	:=el1889s[4,7];	(*裁剪组?单戳纸气缸7基始位*)
stCtrlCylinder[20].DiWorkLimit	:=el1889s[4,8];	(*裁剪组?单戳纸气缸7工作位*)
stCtrlCylinder[21].DiBaseLimit	:=el1889s[4,9];	(*裁剪组?单戳纸气缸8基始位*)
stCtrlCylinder[21].DiWorkLimit	:=el1889s[4,10];	(*裁剪组?单戳纸气缸8工作位*)
stCtrlCylinder[22].DiBaseLimit	:=el1889s[4,11];	(*裁剪组?单戳纸气缸9基始位*)
stCtrlCylinder[22].DiWorkLimit	:=el1889s[4,12];	(*裁剪组?单戳纸气缸9工作位*)
stCtrlCylinder[23].DiBaseLimit	:=el1889s[4,13];	(*裁剪组?单戳纸气缸10基始位*)
stCtrlCylinder[23].DiWorkLimit	:=el1889s[4,14];	(*裁剪组?单戳纸气缸10工作位*)
stCtrlCylinder[24].DiBaseLimit	:=el1889s[4,15];	(*裁剪组?单戳纸气缸11基始位*)
stCtrlCylinder[24].DiWorkLimit	:=el1889s[4,16];	(*裁剪组?单戳纸气缸11工作位*)


(***************************** DI5   ********************************************)
stCtrlCylinder[25].DiBaseLimit	:=el1889s[5,1];	(*裁剪组?单戳纸气缸12基始位*)
stCtrlCylinder[25].DiWorkLimit	:=el1889s[5,2];	(*裁剪组?单戳纸气缸12工作位*)
stCtrlCylinder[26].DiBaseLimit	:=el1889s[5,3];	(*裁剪组?单戳纸气缸13基始位*)
stCtrlCylinder[26].DiWorkLimit	:=el1889s[5,4];	(*裁剪组?单戳纸气缸13工作位*)
stCtrlCylinder[27].DiBaseLimit	:=el1889s[5,5];	(*裁剪组?单戳纸气缸14基始位*)
stCtrlCylinder[27].DiWorkLimit	:=el1889s[5,6];	(*裁剪组?单戳纸气缸14工作位*)
stCtrlCylinder[28].DiBaseLimit	:=el1889s[5,7];	(*裁剪组?单戳纸气缸15基始位*)
stCtrlCylinder[28].DiWorkLimit	:=el1889s[5,8];	(*裁剪组?单戳纸气缸15工作位*)
stCtrlCylinder[29].DiBaseLimit	:=el1889s[5,9];	(*裁剪组?单戳纸气缸16基始位*)
stCtrlCylinder[29].DiWorkLimit	:=el1889s[5,10];	(*裁剪组?单戳纸气缸16工作位*)
stCtrlCylinder[30].DiBaseLimit	:=el1889s[5,11];	(*裁剪组?单戳纸气缸17基始位*)
stCtrlCylinder[30].DiWorkLimit	:=el1889s[5,12];	(*裁剪组?单戳纸气缸17工作位*)
stCtrlCylinder[31].DiBaseLimit	:=el1889s[5,13];	(*裁剪组?单戳纸气缸18基始位*)
stCtrlCylinder[31].DiWorkLimit	:=el1889s[5,14];	(*裁剪组?单戳纸气缸18工作位*)
stCtrlCylinder[32].DiBaseLimit	:=el1889s[5,15];	(*裁剪组?单戳纸气缸19基始位*)
stCtrlCylinder[32].DiWorkLimit	:=el1889s[5,16];	(*裁剪组?单戳纸气缸19工作位*)

(***************************** DI6   ********************************************)
stCtrlCylinder[33].DiBaseLimit	:=el1889s[6,1];	(*裁剪组?单戳纸气缸20基始位*)
stCtrlCylinder[33].DiWorkLimit	:=el1889s[6,2];	(*裁剪组?单戳纸气缸20工作位*)
stCtrlCylinder[34].DiBaseLimit	:=el1889s[6,3];	(*裁剪组?单戳纸气缸21基始位*)
stCtrlCylinder[34].DiWorkLimit	:=el1889s[6,4];	(*裁剪组?单戳纸气缸21工作位*)
stCtrlCylinder[35].DiBaseLimit	:=el1889s[6,5];	(*裁剪组?单戳纸气缸22基始位*)
stCtrlCylinder[35].DiWorkLimit	:=el1889s[6,6];	(*裁剪组?单戳纸气缸22工作位*)
stCtrlCylinder[36].DiBaseLimit	:=el1889s[6,7];	(*裁剪组?单戳纸气缸23基始位*)
stCtrlCylinder[36].DiWorkLimit	:=el1889s[6,8];	(*裁剪组?单戳纸气缸23工作位*)
stCtrlCylinder[37].DiBaseLimit	:=el1889s[6,9];	(*裁剪组?单戳纸气缸24基始位*)
stCtrlCylinder[37].DiWorkLimit	:=el1889s[6,10];	(*裁剪组?单戳纸气缸24工作位*)
stCtrlCylinder[38].DiBaseLimit	:=el1889s[6,11];	(*裁剪组?单戳纸气缸25基始位*)
stCtrlCylinder[38].DiWorkLimit	:=el1889s[6,12];	(*裁剪组?单戳纸气缸25工作位*)


(***************************** DI7   ********************************************)



Axis_Interface[1].Axis_Limit_Pos:=NOT El1889s[7,1]; 	(*模组1正限位*)
Axis_Interface[1].Axis_Limit_Neg:=NOT El1889s[7,2];	(*模组1负限位*)
Axis_Interface[2].Axis_Limit_Pos:=NOT El1889s[7,3];	(*模组2正限位*)
Axis_Interface[2].Axis_Limit_Neg:=NOT El1889s[7,4];	(*模组2负限位*)
Axis_Interface[4].Axis_Limit_Pos:=NOT El1889s[7,5];	(*模组3正限位*)
Axis_Interface[4].Axis_Limit_Neg:=NOT El1889s[7,6];	(*模组3负限位*)
Axis_Interface[3].Axis_Limit_Pos:=NOT El1889s[7,7];	(*模组4正限位*)
Axis_Interface[3].Axis_Limit_Neg:=NOT El1889s[7,8];	(*模组4负限位*)
END_ACTION
ACTION Output:
(***************************** DO1  ********************************************)

El2889s[1,1]	:=	stCtrlCylinder[1].DoAct	;	(*采集组?采集盖下压气缸1?双电控线圈1去工作位*)
El2889s[1,2]	:=	stCtrlCylinder[2].DoAct;		(*采集组?采集盖下压气缸2?双电控线圈1去工作位*)
El2889s[1,3]	:=	stCtrlCylinder[11].DoAct;	(*裁剪组?压板升降气缸?双电控线圈1去工作位*)
El2889s[1,4]	:=	stCtrlCylinder[5].DoAct;		(*气动拧瓶盖组?升降动作?双电控线圈1去工作位*)
El2889s[1,5]	:=	stCtrlCylinder[13].DoAct;	(*裁剪组?防漏气缸去工作位*)
El2889s[1,6]	:=	stCtrlCylinder[12].DoAct;	(*裁剪组?裁剪冲压气缸*)
El2889s[1,7]	:=	stCtrlCylinder[10].DoAct;	(*装盒子组?戳纸升降气缸工作位*)
El2889s[1,8]	:=	stCtrlCylinder[8].DoAct;		(*装盒子组?定位夹紧气缸1工作位*)
El2889s[1,9]	:=	stCtrlCylinder[9].DoAct;		(*装盒子组?定位夹紧气缸2工作位*)
El2889s[1,10]	:=	stCtrlCylinder[7].DoAct;		(*装盒子组?料盒切换动作气缸工作位*)
El2889s[1,11]	:=	stCtrlCylinder[3].DoAct;		(*滤纸转运组吸盘气缸工作位*)
El2889s[1,12]	:=	stCtrlCylinder[4].DoAct;		(*气动拧瓶盖组瓶盖夹爪气缸工作位*)
El2889s[1,13]	:=	stCtrlCylinder[6].DoAct;		(*气动拧瓶盖组 ?水平动作?气缸工作位*)
El2889s[1,14]	:=	stCtrlCylinder[14].DoAct;	(*裁剪组?单戳纸气缸1工作位*)
El2889s[1,15]	:=	stCtrlCylinder[15].DoAct;	(*裁剪组?单戳纸气缸2工作位*)
El2889s[1,16]	:=	stCtrlCylinder[16].DoAct;	(*裁剪组?单戳纸气缸3工作位*)

(***************************** DO2  ********************************************)


El2889s[2,1]	:=	stCtrlCylinder[17].DoAct;		(*裁剪组?单戳纸气缸4工作位*)
El2889s[2,2]	:=	stCtrlCylinder[18].DoAct;		(*裁剪组?单戳纸气缸5工作位*)
El2889s[2,3]	:=	stCtrlCylinder[19].DoAct;		(*裁剪组?单戳纸气缸6工作位*)
El2889s[2,4]	:=	stCtrlCylinder[20].DoAct;		(*裁剪组?单戳纸气缸7工作位*)
El2889s[2,5]	:=	stCtrlCylinder[21].DoAct;		(*裁剪组?单戳纸气缸8工作位*)
El2889s[2,6]	:=	stCtrlCylinder[22].DoAct;		(*裁剪组?单戳纸气缸9工作位*)
El2889s[2,7]	:=	stCtrlCylinder[23].DoAct;		(*裁剪组?单戳纸气缸10工作位*)
El2889s[2,8]	:=	stCtrlCylinder[24].DoAct;		(*裁剪组?单戳纸气缸11工作位*)
El2889s[2,9]	:=	stCtrlCylinder[25].DoAct;		(*裁剪组?单戳纸气缸12工作位*)
El2889s[2,10]	:=	stCtrlCylinder[26].DoAct;		(*裁剪组?单戳纸气缸13工作位*)
El2889s[2,11]	:=	stCtrlCylinder[27].DoAct;		(*裁剪组?单戳纸气缸14工作位*)
El2889s[2,12]	:=	stCtrlCylinder[28].DoAct;		(*裁剪组?单戳纸气缸15工作位*)
El2889s[2,13]	:=	stCtrlCylinder[29].DoAct;		(*裁剪组?单戳纸气缸16工作位*)
El2889s[2,14]	:=	stCtrlCylinder[30].DoAct;		(*裁剪组?单戳纸气缸17工作位*)
El2889s[2,15]	:=	stCtrlCylinder[31].DoAct;		(*裁剪组?单戳纸气缸18工作位*)
El2889s[2,16]	:=	stCtrlCylinder[32].DoAct;		(*裁剪组?单戳纸气缸19工作位*)

(***************************** DO3  ********************************************)


El2889s[3,1]	:=	stCtrlCylinder[33].DoAct;		(*裁剪组?单戳纸气缸20工作位*)
El2889s[3,2]	:=	stCtrlCylinder[34].DoAct;		(*裁剪组?单戳纸气缸21工作位*)
El2889s[3,3]	:=	stCtrlCylinder[35].DoAct;		(*裁剪组?单戳纸气缸22工作位*)
El2889s[3,4]	:=	stCtrlCylinder[36].DoAct;		(*裁剪组?单戳纸气缸23工作位*)
El2889s[3,5]	:=	stCtrlCylinder[37].DoAct;		(*裁剪组?单戳纸气缸24工作位*)
El2889s[3,6]	:=	stCtrlCylinder[38].DoAct;		(*裁剪组?单戳纸气缸25工作位*)


El2889s[3,9]	:=	stMachine.boBtnStartLed;(*启动按钮灯*)
El2889s[3,10]	:=	stMachine.	boLamp_Red		(*灯柱-红*);
El2889s[3,11]	:=	stMachine.	boLamp_Yellow		(*灯柱-黄*);
El2889s[3,12]	:=	stMachine.boBtnStopLed;		(*急停按钮灯*)

El2889s[3,13]	:=	NOT stCtrlCylinder[1].DoAct;		(*采集组?采集盖下压气缸1?双电控线圈2基始位*)
El2889s[3,14]	:=	NOT stCtrlCylinder[2].DoAct;		(*采集组?采集盖下压气缸2?双电控线圈2基始位*)
El2889s[3,15]	:=	NOT stCtrlCylinder[11].DoAct;	(*裁剪组?压板升降气缸基始位*)
El2889s[3,16]	:=	NOT stCtrlCylinder[5].DoAct;		(*气动拧瓶盖组?升降动作气缸基始位*)
END_ACTION

(* POU 01_IO/Aifilter, ST *)
FUNCTION_BLOCK Aifilter
VAR_INPUT
	vi_Filter:REAL;
	n:UINT:=10;
END_VAR
VAR_OUTPUT
	vo_Filter:REAL;
END_VAR
VAR
	Filter	:ARRAY[1..100] OF REAL;
	Sum:REAL;
	i:UINT;
	counter:INT;
END_VAR
counter:=counter+1;
n:=LIMIT(5,n,100);
IF counter>=10 THEN
	MEMCPY(ADR(Filter[1]),ADR(Filter[2]),SIZEOF(Filter[1])*(n-1));
	Filter[n]:=vi_Filter;
	sum:=0;
	FOR  i:=1 TO n DO
		sum:=sum+Filter[i];
	END_FOR
	vo_Filter:=sum/n;
	counter:=0;
END_IF
END_FUNCTION_BLOCK

(* POU 02_Common/PRG_Alarm, ST *)
PROGRAM PRG_Alarm
VAR
	i: UINT;
	iNc:UINT;
	iDr:UINT;
	tDelay	:ARRAY[1..MaxAlarms]OF TON;
	counter: UINT;
	bDelayFlag: BOOL;
	tDelayReset:TON;
END_VAR
ActAlarm;
ActWarning;
Act_Alarm_Modbus;
Act_Warm_Modbus;

bGlobalErrorMark:=FALSE;
FOR i:=1 TO MaxAlarms DO
(*任何一个报警触发时，都会触发报警  并且锁住*)
	IF I<>26 THEN
	bGlobalErrorMark:=bGlobalErrorMark OR arrAlarm[i];
	END_IF
END_FOR

tDelayReset(IN:=NOT tDelayReset.Q  , PT:=t#10s , Q=> , ET=> );

IF bSysReset OR tDelayReset.Q  THEN
	PRG_Alarm.Act_ResetAlarm();
END_IF

tDelayReset(IN:=NOT tDelayReset.Q  , PT:=t#10s , Q=> , ET=> );

MSGList1_Alarm:=FALSE;
FOR i:=1 TO MaxAlarms DO
(*任何一个报警触发时，都会触发报警  并且锁住*)
	MSGList1_Alarm:=MSGList1_Alarm OR MSGList1[i];
END_FOR
END_PROGRAM
ACTION Act_Alarm_Modbus:
iAlarmNetConnect.0:=arrAlarm[21];
iAlarmNetConnect.1:=arrAlarm[22];
iAlarmNetConnect.2:=arrAlarm[23];
iAlarmNetConnect.3:=arrAlarm[24];
iAlarmNetConnect.4:=arrAlarm[25];
iAlarmNetConnect.5:=arrAlarm[26];
iAlarmNetConnect.6:=arrAlarm[27];
iAlarmNetConnect.7:=arrAlarm[28];
END_ACTION
ACTION Act_ResetAlarm:
MEMSET(ADR(arrAlarm),0,SIZEOF(arrAlarm));
MEMSET(ADR(arrWarning),0,SIZEOF(arrWarning));


bAxisMovingAbsAlarm[1]:=FALSE;
bAxisMovingAbsAlarm[2]:=FALSE;
bAxisMovingAbsAlarm[3]:=FALSE;
bAxisMovingAbsAlarm[4]:=FALSE;
bAxisMovingAbsAlarm[5]:=FALSE;

bAxisMovingAbsAlarm[6]:=FALSE;
bAxisMovingAbsAlarm[7]:=FALSE;
bAxisMovingAbsAlarm[8]:=FALSE;
bAxisMovingAbsAlarm[9]:=FALSE;
bAxisMovingAbsAlarm[10]:=FALSE;
bAxisMovingAbsAlarm[11]:=FALSE;
bAxisMovingAbsAlarm[12]:=FALSE;
bAxisMovingAbsAlarm[13]:=FALSE;
bAxisMovingAbsAlarm[14]:=FALSE;
END_ACTION
ACTION Act_Warm_Modbus:
iWarnMoveAbs.0:=arrWarning[1];
iWarnMoveAbs.1:=arrWarning[2];
iWarnMoveAbs.2:=arrWarning[3];
iWarnMoveAbs.3:=arrWarning[4];
iWarnMoveAbs.4:=arrWarning[5];
iWarnMoveAbs.5:=arrWarning[6];
iWarnMoveAbs.6:=arrWarning[7];
iWarnMoveAbs.7:=arrWarning[8];
iWarnMoveAbs.8:=arrWarning[9];
iWarnMoveAbs.9:=arrWarning[10];
iWarnMoveAbs.10:=arrWarning[11];
iWarnMoveAbs.11:=arrWarning[12];
iWarnMoveAbs.12:=arrWarning[13];
iWarnMoveAbs.13:=arrWarning[14];
iWarnMoveAbs.14:=arrWarning[15];
iWarnMoveAbs.15:=arrWarning[16];
END_ACTION
ACTION ActAlarm:
IF bDelayFlag THEN
(*急停报警*)
	IF NOT arrAlarm[1]
	THEN
		arrAlarm[1]:=bSysEstop;
	END_IF


(*轴类相关报警*)

	FOR i:=1 TO 5 BY 1 DO
		IF axisarr[i].Status.Error THEN
			arrAlarm[i+11]:=TRUE;		(*轴报警，含虚拟轴*)
		END_IF
		IF i<>5 THEN
			IF Axis_Interface[i].Axis_Limit_pos THEN
				arrAlarm[i+30]:=TRUE;	(*轴的限位报警*)
			END_IF
			IF Axis_Interface[i].Axis_Limit_neg THEN
				arrAlarm[i+1]:=TRUE;
			END_IF
		END_IF
	END_FOR

	FOR i:=1 TO NumOfDrives DO
		IF ( DrivesOP[i]<>iEcatOp) THEN
			arrAlarm[i+20]:=TRUE;
		END_IF
	END_FOR
END_IF
(*PLC周期是2MS，累加3500个周期，就是延迟7秒后，给出网报警*)
IF counter>3500 THEN
	bDelayFlag:=TRUE;
	(*counter:=0;*)
END_IF

IF NOT bDelayFlag THEN
	counter:=counter+1;
END_IF
END_ACTION
ACTION ActWarning:
;
(*在judgement程序中给出了警告的赋值*)


(*模组1X轴走定位超过2S不动，警告*)
IF bAxisMovingAbsAlarm[1] THEN
	arrWarning[1]:=TRUE;
END_IF


(*模组2Z轴走定位超过2S不动，警告*)
IF bAxisMovingAbsAlarm[2] THEN
	arrWarning[2]:=TRUE;
END_IF


(*模组3X轴走定位超过2S不动，警告*)
IF bAxisMovingAbsAlarm[3] THEN
	arrWarning[3]:=TRUE;
END_IF


(*模组4Y轴走定位超过2S不动，警告*)
IF bAxisMovingAbsAlarm[4] THEN
	arrWarning[4]:=TRUE;
END_IF


(*模组5旋转轴走定位超过2S不动，警告*)
IF bAxisMovingAbsAlarm[5] THEN
	arrWarning[5]:=TRUE;
END_IF

(*切换到自动模式之前，请先执行去准备位*)
IF NOT bAutoReady AND bSwitchAutoMode THEN
	arrWarning[15]:=TRUE;
END_IF

(*去准备位之前，请先执行回原*)
IF NOT All_Homed_OK AND bGoPrepareAuto THEN
	arrWarning[16]:=TRUE;
END_IF
END_ACTION

(* POU 03_机台/00_通用/PRG_Monitor, ST *)
PROGRAM PRG_Monitor
VAR
	iDrive	:UINT;
	i: UINT;
END_VAR
(*系统需要进行某一步之前需要对一些关键状态进行判定*)

bDeviceStateOK:=TRUE;
bDriveModeOK:=TRUE;
(*
FOR iDrive:=1 TO NumOfDrives DO
	bDeviceStateOK:=bDeviceStateOK AND DrivesOP[iDrive]=iEcatOp;
	bDriveModeOK:=bDriveModeOK AND (iActDriveMode[iDrive]=iSetDriveMode[iDrive]);
END_FOR

*)
END_PROGRAM

(* POU 06_自动/PRG_Auto, ST *)
PROGRAM PRG_Auto
VAR
	eRuningStep				:	UINT;
	eStopStep				:	UINT;

	trAutoRuning:R_TRIG;
	tResetAutoSignal:TON;

(*trigers*)
	rTrigGlobalError			:	R_TRIG;	(*需要停机的错误，触发后不退出自动，复位错误后，可以继续运行*)
	rTrigEstop				:	R_TRIG;	(*需要停机，并且完成后进入急停*)
	rTrigstop				:	R_TRIG;(*需要停机，停完后，点启动可以继续跑*)
	rTrigSwitchManual		:	R_TRIG;	(*需要停机，停完后切到手动*)
	rTrigStart				:	R_TRIG;	(*启动*)

(*delay*)
	tStopDelay	:TON;

	fbHaltMain: MC_Halt;
	fbMoveMain: MC_MoveRelative;
	fTempDistanceInCycle_L: REAL;
	fTempDistanceInCycle_R: REAL;
	fRecordMainPos: REAL;
	iTest400: UINT;
	iTest500: UINT;
	itest1: UINT:=0;
	itest2:	UINT:=0;
	itest3:	UINT:=0;
	itest4:	UINT:=0;

(****************************Modbus_TCP*******************************)
	iXStep1: UINT;
	iXStep2: UINT;
	iZStep1: UINT;
	iZStep2: UINT;

	iX2Step1: UINT;
	iX2Step2: UINT;
	iY2Step1: UINT;
	iY2Step2: UINT;

	iRStep1: UINT;
	iRStep2: UINT;
	iRStep3: UINT;
	iRStep4: UINT;
	iHorizontalStep1: UINT;
	iHorizontalStep2: UINT;
	iRotaryStep1: UINT;
	iRotaryStep2: UINT;
	iCollimationStep1:UINT;
	iCollimationStep2:UINT;

	fPos_X_Axis:REAL;
	fPos_Z_Axis:REAL;


	fPos_X2_Axis:REAL;
	fPos_Y2_Axis:REAL;

	fPos_R_Axis:REAL;
	fPos_CollimationAxis:REAL;


	fPos_HorizontalAxis:REAL;
	fPos_RotaryAxis:REAL;

	rPutPermit_Cmd:R_TRIG;
	rGetPermit_Cmd:R_TRIG;
	iPutStep:UINT;
	iGetStep:UINT;

	tDelayMC_AbsAlarm:ARRAY[1..20] OF TON;
	r_TRIG_Cmd:ARRAY[1..20] OF R_TRIG;

	bX_Axis_Abs: BOOL;
	bX_Axis_Stop: BOOL;
	bZ_Axis_Abs: BOOL;
	bZ_Axis_Stop: BOOL;

	bX2_Axis_Abs: BOOL;
	bX2_Axis_Stop: BOOL;
	bY2_Axis_Abs: BOOL;
	bY2_Axis_Stop: BOOL;

	bR_Axis_Abs: BOOL;
	bR_Axis_Stop: BOOL;
	bHorizontal_Axis_Abs: BOOL;
	bHorizontal_Axis_Stop: BOOL;
	bRotary_Axis_Abs: BOOL;
	bRotary_Axis_Stop: BOOL;
	bCollimationAxis_Abs: BOOL;
	bCollimationAxis_Stop: BOOL;

	bR_Axis_Velo: BOOL;
	bR_Axis_Stop1: BOOL;
END_VAR
IF bSysReset THEN
	bStopFinished:=FALSE;
END_IF

bAutoModeRunning:=(eRuningStep>0);	(*切出自动时，会先把eRuningStep置为0*)
END_PROGRAM
ACTION Act_Modbus_TCP:
fPos_X_Axis:=iPos_X_Axis*0.1;	(*模组1X轴电机*)
fPos_Z_Axis:=iPos_Z_Axis*0.1;	(*模组2Z轴电机*)

fPos_X2_Axis:=iPos_X2_Axis*0.1;	(*模组3X轴电机*)
fPos_Y2_Axis:=iPos_Y2_Axis*0.1;	(*模组4Y轴电机*)


fPos_R_Axis:=iPos_R_Axis*0.1;	(*旋转电机*)

(*模组1X轴电机*)
CASE iX_Axis_Cmd OF
0:
	bX_Axis_Abs:=FALSE;
	bX_Axis_Stop:=FALSE;
1:
	bX_Axis_Abs:=TRUE;
2:
	bX_Axis_Stop:=TRUE;
END_CASE

r_TRIG_Cmd[1](CLK:=bX_Axis_Abs , Q=> );

	CASE iXStep1 OF
	0:
		IF r_TRIG_Cmd[1].Q THEN
			iXStep1:=5;
			Axis_Interface[1].bMoveAbs:=FALSE;
		END_IF
	5:
		IF ABS(fPos_X_Axis-Axis_Interface[1].fActPos)>0.1  THEN
			iXStep1:=10;
			iXStep2:=0;
			Axis_Interface[1].bStop:=FALSE;
			tDelayMC_AbsAlarm[1](in:=FALSE);
		ELSE
			iXStep1:=0;
		END_IF
	10:			(*工作节拍*)
		Axis_Interface[1].fPositon_of_Abs:=fPos_X_Axis;
		Axis_Interface[1].fVelocity_of_Abs:=stAxisParam[1].fVelo_of_Auto;
		Axis_Interface[1].bMoveAbs:=TRUE;
		IF ABS(Axis_Interface[1].fActPos-fPos_X_Axis)<0.1 AND ABS(Axis_Interface[1].fActVelo)<0.1 THEN
			iXStep1:=50;
		END_IF
		Axis_Interface[1].bMoveAbs:=(iXStep1=10);
		tDelayMC_AbsAlarm[1](IN:=Axis_Interface[1].Axis_NotMoving , PT:=t#2s , Q=> , ET=> );
		IF tDelayMC_AbsAlarm[1].Q THEN
			bAxisMovingAbsAlarm[1]:=TRUE;
			iXStep1:=50;
		END_IF
	50:
		iXStep1:=0;
		tDelayMC_AbsAlarm[1](in:=FALSE);
	END_CASE


r_TRIG_Cmd[2](CLK:=bX_Axis_Stop , Q=> );
	CASE iXStep2 OF
	0:
		IF r_TRIG_Cmd[2].Q THEN
			iXStep2:=5;
		END_IF

	5:
		IF NOT Axis_Interface[1].Axis_NotMoving THEN
			iXStep2:=10;
			iXStep1:=0;
			Axis_Interface[1].bMoveAbs:=FALSE;
		ELSE
			iXStep2:=0;
		END_IF
	10:
		Axis_Interface[1].bStop:=TRUE;
		iXStep2:=50;
	50:
		IF Axis_Interface[1].Axis_NotMoving THEN
			iXStep2:=0;
			Axis_Interface[1].bStop:=FALSE;
		END_IF
	END_CASE


(*模组1Z轴电机*)

CASE iZ_Axis_Cmd OF
0:
	bZ_Axis_Abs:=FALSE;
	bZ_Axis_Stop:=FALSE;
1:
	bZ_Axis_Abs:=TRUE;
2:
	bZ_Axis_Stop:=TRUE;
END_CASE

r_TRIG_Cmd[3](CLK:=bZ_Axis_Abs , Q=> );
	CASE iZStep1 OF
	0:
		IF r_TRIG_Cmd[3].Q THEN
			iZStep1:=5;
		END_IF

	5:
		IF ABS(fPos_Z_Axis-Axis_Interface[2].fActPos)>0.1  THEN
			iZStep1:=10;
			iZStep2:=0;
			Axis_Interface[2].bStop:=FALSE;
			tDelayMC_AbsAlarm[2](in:=FALSE);
		ELSE
			iZStep1:=0;
		END_IF
	10:
		Axis_Interface[2].fPositon_of_Abs:=fPos_Z_Axis;
		Axis_Interface[2].fVelocity_of_Abs:=stAxisParam[2].fVelo_of_Auto;
		Axis_Interface[2].bMoveAbs:=TRUE;
		IF ABS(Axis_Interface[2].fActPos-fPos_Z_Axis)<0.1 AND ABS(Axis_Interface[2].fActVelo)<0.1 THEN
			iZStep1:=50;
		END_IF
		Axis_Interface[2].bMoveAbs:=(iZStep1=10);
		tDelayMC_AbsAlarm[2](IN:=Axis_Interface[2].Axis_NotMoving , PT:=t#2s , Q=> , ET=> );
		IF tDelayMC_AbsAlarm[2].Q THEN
			bAxisMovingAbsAlarm[2]:=TRUE;
			iZStep1:=50;
		END_IF
	50:
		iZStep1:=0;
		tDelayMC_AbsAlarm[2](in:=FALSE);
	END_CASE

r_TRIG_Cmd[4](CLK:=bZ_Axis_Stop , Q=> );
	CASE iZStep2 OF
	0:
		IF r_TRIG_Cmd[4].Q THEN
			iZStep2:=5;
		END_IF
	5:
		IF NOT Axis_Interface[2].Axis_NotMoving THEN
			iZStep2:=10;
			iZStep1:=0;
			Axis_Interface[2].bMoveAbs:=FALSE;
		ELSE
			iZStep2:=0;
		END_IF
	10:
		Axis_Interface[2].bStop:=TRUE;
		iZStep2:=50;
	50:
		IF Axis_Interface[2].Axis_NotMoving THEN
			iZStep2:=0;
			Axis_Interface[2].bStop:=FALSE;
		END_IF
	END_CASE



(*模组3X轴电机*)
CASE iX2_Axis_Cmd OF
0:
	bX2_Axis_Abs:=FALSE;
	bX2_Axis_Stop:=FALSE;
1:
	bX2_Axis_Abs:=TRUE;
2:
	bX2_Axis_Stop:=TRUE;
END_CASE

r_TRIG_Cmd[5](CLK:=bX2_Axis_Abs , Q=> );

	CASE iX2Step1 OF
	0:
		IF r_TRIG_Cmd[5].Q THEN
			iX2Step1:=5;
			Axis_Interface[3].bMoveAbs:=FALSE;
		END_IF
	5:
		IF ABS(fPos_X2_Axis-Axis_Interface[3].fActPos)>0.1  THEN
			iX2Step1:=10;
			iX2Step2:=0;
			Axis_Interface[3].bStop:=FALSE;
			tDelayMC_AbsAlarm[3](in:=FALSE);
		ELSE
			iX2Step1:=0;
		END_IF
	10:			(*工作节拍*)
		Axis_Interface[3].fPositon_of_Abs:=fPos_X2_Axis;
		Axis_Interface[3].fVelocity_of_Abs:=stAxisParam[3].fVelo_of_Auto;
		Axis_Interface[3].bMoveAbs:=TRUE;
		IF ABS(Axis_Interface[3].fActPos-fPos_X2_Axis)<0.1 AND ABS(Axis_Interface[3].fActVelo)<0.1 THEN
			iX2Step1:=50;
		END_IF
		Axis_Interface[3].bMoveAbs:=(iX2Step1=10);
		tDelayMC_AbsAlarm[3](IN:=Axis_Interface[3].Axis_NotMoving , PT:=t#2s , Q=> , ET=> );
		IF tDelayMC_AbsAlarm[3].Q THEN
			bAxisMovingAbsAlarm[3]:=TRUE;
			iX2Step1:=50;
		END_IF
	50:
		iX2Step1:=0;
		tDelayMC_AbsAlarm[3](in:=FALSE);
	END_CASE

r_TRIG_Cmd[6](CLK:=bX2_Axis_Stop , Q=> );
	CASE iX2Step2 OF
	0:
		IF r_TRIG_Cmd[6].Q THEN
			iX2Step2:=5;
		END_IF

	5:
		IF NOT Axis_Interface[3].Axis_NotMoving THEN
			iX2Step2:=10;
			iX2Step1:=0;
			Axis_Interface[3].bMoveAbs:=FALSE;
		ELSE
			iX2Step2:=0;
		END_IF
	10:
		Axis_Interface[3].bStop:=TRUE;
		iX2Step2:=50;
	50:
		IF Axis_Interface[3].Axis_NotMoving THEN
			iX2Step2:=0;
			Axis_Interface[3].bStop:=FALSE;
		END_IF
	END_CASE


(*模组4Y轴电机*)

CASE iY2_Axis_Cmd OF
0:
	bY2_Axis_Abs:=FALSE;
	bY2_Axis_Stop:=FALSE;
1:
	bY2_Axis_Abs:=TRUE;
2:
	bY2_Axis_Stop:=TRUE;
END_CASE

r_TRIG_Cmd[7](CLK:=bY2_Axis_Abs , Q=> );
	CASE iY2Step1 OF
	0:
		IF r_TRIG_Cmd[7].Q THEN
			iY2Step1:=5;
		END_IF

	5:
		IF ABS(fPos_Y2_Axis-Axis_Interface[4].fActPos)>0.1  THEN
			iY2Step1:=10;
			iY2Step2:=0;
			Axis_Interface[4].bStop:=FALSE;
			tDelayMC_AbsAlarm[4](in:=FALSE);
		ELSE
			iY2Step1:=0;
		END_IF
	10:
		Axis_Interface[4].fPositon_of_Abs:=fPos_Y2_Axis;
		Axis_Interface[4].fVelocity_of_Abs:=stAxisParam[4].fVelo_of_Auto;
		Axis_Interface[4].bMoveAbs:=TRUE;
		IF ABS(Axis_Interface[4].fActPos-fPos_Y2_Axis)<0.1 AND ABS(Axis_Interface[4].fActVelo)<0.1 THEN
			iY2Step1:=50;
		END_IF
		Axis_Interface[4].bMoveAbs:=(iY2Step1=10);
		tDelayMC_AbsAlarm[4](IN:=Axis_Interface[4].Axis_NotMoving , PT:=t#2s , Q=> , ET=> );
		IF tDelayMC_AbsAlarm[4].Q THEN
			bAxisMovingAbsAlarm[4]:=TRUE;
			iY2Step1:=50;
		END_IF
	50:
		iY2Step1:=0;
		tDelayMC_AbsAlarm[4](in:=FALSE);
	END_CASE

r_TRIG_Cmd[8](CLK:=bY2_Axis_Stop , Q=> );
	CASE iY2Step2 OF
	0:
		IF r_TRIG_Cmd[8].Q THEN
			iY2Step2:=5;
		END_IF
	5:
		IF NOT Axis_Interface[4].Axis_NotMoving THEN
			iY2Step2:=10;
			iY2Step1:=0;
			Axis_Interface[4].bMoveAbs:=FALSE;
		ELSE
			iY2Step2:=0;
		END_IF
	10:
		Axis_Interface[4].bStop:=TRUE;
		iY2Step2:=50;
	50:
		IF Axis_Interface[4].Axis_NotMoving THEN
			iY2Step2:=0;
			Axis_Interface[4].bStop:=FALSE;
		END_IF
	END_CASE


(*旋转电机*)
CASE iR_Axis_Cmd OF
0:
	bR_Axis_Abs:=FALSE;
	bR_Axis_Stop:=FALSE;
1:
	bR_Axis_Abs:=TRUE;
2:
	bR_Axis_Stop:=TRUE;
END_CASE

r_TRIG_Cmd[9](CLK:=bR_Axis_Abs , Q=> );
	CASE iRStep1 OF
	0:
		IF r_TRIG_Cmd[9].Q THEN
			iRStep1:=5;
			Axis_Interface[5].bMoveAbs:=FALSE;
		END_IF

	5:
		IF ABS(fPos_R_Axis-Axis_Interface[5].fActPos)>0.1  THEN
			iRStep1:=10;
			iRStep2:=0;
			Axis_Interface[5].bStop:=FALSE;
			tDelayMC_AbsAlarm[5](in:=FALSE);
		ELSE
			iRStep1:=0;
		END_IF
	10:
		Axis_Interface[5].fPositon_of_Abs:=fPos_R_Axis;
		Axis_Interface[5].fVelocity_of_Abs:=stAxisParam[5].fVelo_of_Auto;
		Axis_Interface[5].bMoveAbs:=TRUE;
		IF ABS(Axis_Interface[5].fActPos-fPos_R_Axis)<0.1 AND ABS(Axis_Interface[5].fActVelo)<0.1 THEN
			iRStep1:=50;
		END_IF
		Axis_Interface[5].bMoveAbs:=(iRStep1=10);
		tDelayMC_AbsAlarm[5](IN:=Axis_Interface[5].Axis_NotMoving , PT:=t#2s , Q=> , ET=> );
		IF tDelayMC_AbsAlarm[5].Q THEN
			bAxisMovingAbsAlarm[5]:=TRUE;
			iRStep1:=50;
		END_IF
	50:
		iRStep1:=0;
		tDelayMC_AbsAlarm[5](in:=FALSE);
	END_CASE

r_TRIG_Cmd[10](CLK:=bR_Axis_Stop , Q=> );
	CASE iRStep2 OF
	0:
		IF r_TRIG_Cmd[10].Q THEN
			iRStep2:=5;
		END_IF

	5:
		IF NOT Axis_Interface[5].Axis_NotMoving THEN
			iRStep2:=10;
			iRStep1:=0;
			Axis_Interface[5].bMoveAbs:=FALSE;
		ELSE
			iRStep2:=0;
		END_IF
	10:
		Axis_Interface[5].bStop:=TRUE;
		iRStep2:=50;
	50:
		IF Axis_Interface[5].Axis_NotMoving THEN
			iRStep2:=0;
			Axis_Interface[5].bStop:=FALSE;
		END_IF
	END_CASE




(*一键回原*)
CASE iGoHomeTogether_Cmd OF
0:
	bGoHomeTogether_Cmd:=FALSE;
1:
	bGoHomeTogether_Cmd:=TRUE;
2:
	bGoHomeTogether_Cmd:=FALSE;
END_CASE

(*一键去准备位*)
CASE iGoPrepareAuto_Cmd OF
0:
	bGoPrepareAuto_Cmd:=FALSE;
1:
	bGoPrepareAuto_Cmd:=TRUE;
2:
	bGoPrepareAuto_Cmd:=FALSE;
END_CASE


(*自动切换*)

CASE iAuto_Cmd OF
0:
	bAuto_Cmd:=FALSE;
1:
	bAuto_Cmd:=FALSE;
2:
	bAuto_Cmd:=TRUE;
END_CASE
END_ACTION
ACTION Act_Run:
CASE eRuningStep OF
0:
	IF bSysStart AND bAutoReady THEN		(*bAutoReady会在手动模式进行判断*)
		eRuningStep:=100;
		bStopFinished:=TRUE;
	END_IF
100:
	IF bSysStop  THEN
		eRuningStep:=200;
	END_IF
200:(*要把TCP的程序执行完，才能推出自动程序*)
	IF iXStep1=0 AND iXStep2=0 AND iZStep1=0 AND iZStep2=0 AND iX2Step1=0 AND iX2Step2=0 AND iY2Step1=0 AND iY2Step2=0 AND iRstep1 = 0 AND iRstep2=0
THEN
		eRuningStep:=0;
		bStopFinished:=FALSE;
	END_IF

END_CASE
END_ACTION

(* POU 03_机台/00_通用/PRG_Power, ST *)
PROGRAM PRG_Power
(*本设置只是在上电初始化时设定一次，需要实时改变的值，需要在其他程序中赋值*)
(*急停复位也会重新执行一次，由于会断使能，所以普通报错不要跳入*)

VAR
	i: UINT;
END_VAR
(*****************************检查UPS以及接触器等回路信号*************************)

;
(***********************************驱动器控制模式设定*************************)
(*倍福驱动器不用设置模式*)
(*
FOR i:=1 TO NumOfDrives-2 DO
	iSetDriveMode[i]:=CSP;
END_FOR

iSetDriveMode[9]:=
iSetDriveMode[10]:=CST;		(*9,10号轴力矩模式*)
*)

(***********************************步进电机设定*************************)
(*
(*设定步进驱动器的峰值电流为mA*)
iSetPeakCurrent:=6000;
*)

(***********************************手动按钮，自动指令，内部指令的清零*************************)

FOR i:=1 TO MaxAxes DO
(*使能*)
	Axis_Interface[i].bEnable:=FALSE;
	Axis_Interface[i].bEnableFw:=FALSE;
	Axis_Interface[i].bEnableBw:=FALSE;
(*可以根据工艺要求，取消一部分轴的断使能 20210529 sheniang*)

(*其他操作指令*)
	Axis_Interface[i].bHome:=FALSE;
	Axis_Interface[i].bJog_Bw:=FALSE;
	Axis_Interface[i].bHalt:=FALSE;
	Axis_Interface[i].bJog_Fw:=FALSE;
	Axis_Interface[i].bMoveAbs:=FALSE;
	Axis_Interface[i].bMoveVelo:=FALSE;
	Axis_Interface[i].bMoveRel:=FALSE;
	Axis_Interface[i].bReset:=FALSE;
	Axis_Interface[i].bStop:=FALSE;
	Axis_Interface[i].bGearOut:=FALSE;
	Axis_Interface[i].bGearIn:=FALSE;
	Axis_Interface[i].bSetPos:=FALSE;
	Axis_Interface[i].fOverride:=100;

END_FOR

bHasResetOnce:=FALSE;
END_PROGRAM

(* POU 03_机台/00_通用/PRG_ServOn, ST *)
PROGRAM PRG_ServOn
(**专门处理使能的程序，因为不一定只在初始化时使用，所以从初始化程序中脱离开来**)
VAR
	i: UINT;
	Encoder: BOOL;
END_VAR
(*使能*)
FOR i:=1 TO MaxAxes DO
	Axis_Interface[i].bEnable:=TRUE;
	Axis_Interface[i].bEnableFw:=TRUE;
	Axis_Interface[i].bEnableBw:=TRUE;
END_FOR
END_PROGRAM

(* POU 03_机台/00_通用/PRG_Init, ST *)
PROGRAM PRG_Init
(**处理除了使能以外的程序**)
VAR
	i:UINT;
	bNomoreTest: BOOL;
END_VAR
(*在进入手动前执行一次*)

FOR i:=1 TO MaxAxes BY 1 DO
	stHmiAxisCmd[i].bEnable:=TRUE;				(*进入手动后，使能会由stAxisCmd控制，防止使能自动掉，所以给一次true*)
	stHmiAxisCmd[i].bHome:=FALSE;
	stHmiAxisCmd[i].bJog_Bw:=FALSE;
	stHmiAxisCmd[i].bJog_Fw:=FALSE;
END_FOR
END_PROGRAM

(* POU 05_手动/PRG_Manual, ST *)
PROGRAM PRG_Manual
VAR
	i: UINT;
	fbJogMaster: MC_Jog;

	tDancerSetPos	:TON;

	fLeftRollDiam_1: REAL;
	fRightRollDiam_1: REAL;
	iStep: INT;
	iStep1: INT;
	rtMoveAbs			: ARRAY[1..MaxAxes] OF  R_TRIG;
	ftMoveAbs			: ARRAY[1..MaxAxes] OF  F_TRIG;
	rtHome1			: R_TRIG;
	rtHome2			:R_TRIG;
	ftHome1			: F_TRIG;
	ftHome2			:F_TRIG;
	rtEnable			: ARRAY[1..MaxAxes] OF  R_TRIG;
	ftEnable			: ARRAY[1..MaxAxes] OF  F_TRIG;
	Rtrig_HMI_SetButton:ARRAY[1..5] OF R_TRIG;
	Ftrig_HMI_SetButton:ARRAY[1..5] OF F_TRIG;
	AxisSetTim:ARRAY[1..5] OF TON;

	rtAxisHome			: ARRAY[1..MaxAxes] OF  R_TRIG;
	ftAxisHome			: ARRAY[1..MaxAxes] OF  F_TRIG;

END_VAR
(*一键回参*)
PRG_GoHomeTogether();

(*一键准备功能*)

PRG_AutoPreparation();

(*回原点*)
FOR i:=1 TO NumOfDrives DO
		rtAxisHome[I](CLK:=stHmiAxisCmd[i].bHome);
		IF rtAxisHome[I].Q AND ABS(Axis_Interface[i].fActPos)>0.1 THEN
			Axis_Interface[i].bMoveAbs:=TRUE ;
			Axis_Interface[i].fPositon_of_Abs:=0  ;
			Axis_Interface[i].fVelocity_of_Abs:=stAxisParam[i].fVelo_of_Posi;
		END_IF
		ftAxisHome[I](CLK:=stHmiAxisCmd[i].bHome);
		IF ftAxisHome[I].Q THEN
			Axis_Interface[i].bMoveAbs:=FALSE ;
		END_IF
END_FOR


(*手动定位*)

FOR i:=1 TO NumOfDrives DO
	rtMoveAbs[i](CLK:=stHmiAxisCmd[i].bMoveAbs , Q=> );
	IF rtMoveAbs[i].Q THEN
		Axis_Interface[i].bMoveAbs:=TRUE ;
		Axis_Interface[i].fPositon_of_Abs:=stAxisParam[i].fTargetPosi  ;		(*手动触发的定位，自然会置false*)
	END_IF
	ftMoveAbs[i](CLK:=stHmiAxisCmd[i].bMoveAbs , Q=> );
	IF ftMoveAbs[i].Q THEN
		Axis_Interface[i].bMoveAbs:=FALSE ;
	END_IF
	Axis_Interface[i].fVelocity_of_Abs:=stAxisParam[i].fVelo_of_Posi;

	CASE stAxisParam[i].iTargetNr OF
		0:stAxisParam[i].fTargetPosi:= stAxisParam[i].StandbyPos;(*待机位*)
		1:stAxisParam[i].fTargetPosi:= stAxisParam[i].WorkPos1;
		2:stAxisParam[i].fTargetPosi:= stAxisParam[i].WorkPos2;
		3:stAxisParam[i].fTargetPosi:= stAxisParam[i].WorkPos3;
	END_CASE

END_FOR

(*设置原点*)
FOR i:=1 TO 5 DO
	Rtrig_HMI_SetButton[i](CLK:=stHmiAxisCmd[I].bSetBiasBnt, Q=> );
	Ftrig_HMI_SetButton[i](CLK:=stHmiAxisCmd[I].bSetBiasBnt, Q=> );
	IF Rtrig_HMI_SetButton[I].Q THEN
		fSaveBias[I]:=fSaveBias[I]+AxisArr[I].NcToPlc.ActPos;
	END_IF
	IF Ftrig_HMI_SetButton[i].Q THEN
		Axis_Interface[i].fPosition_ToBeSet :=-0;
		Axis_Interface[i].bSetPos:=TRUE;(*触发信号*)
	END_IF
	AxisSetTim[i](IN:= Axis_Interface[i].bSetPos, PT:=t#0.1s , Q=> , ET=> );
	IF AxisSetTim[i].Q THEN
		Axis_Interface[i].bSetPos:=FALSE ;
		AxisSetTim[i] (IN:=FALSE , PT:=t#0.1s, Q=> , ET=> );
	END_IF
END_FOR
END_PROGRAM

(* POU 03_机台/01_一键回原/PRG_GoHomeTogether, ST *)
PROGRAM PRG_GoHomeTogether
VAR
	i: UINT;
	iPullAxisHomeStep: INT;
	rTrig:R_TRIG;
	iStep:UINT;
	bAxisNotMoving:BOOL;
	tDelay:TON;
END_VAR
(***************************** 物理回参   ********************************************)
rTrig(CLK:=bGoHomeTogether OR bGoHomeTogether_Cmd, Q=> );

(*************************回参完成信号的判定***************************)
CASE iStep OF
0:
	IF rTrig.Q THEN
		iStep:=100;
		All_Homed_OK:=FALSE;
		bAutoReady:=FALSE;
	END_IF
100:
	FOR i:=1 TO NumOfCylinders DO
		stCtrlCylinder[i].bBack:=TRUE;	(*气缸回原*)
	END_FOR
	IF bAllCylinderBase THEN
		iStep:=110;
	END_IF
110:
	FOR i:=MinHomeAxis TO MaxHomeAxis DO
		Axis_Interface[i].bMoveAbs:=TRUE ;
		Axis_Interface[i].fPositon_of_Abs:=0  ;
		Axis_Interface[i].fVelocity_of_Abs:=stAxisParam[i].fVelo_of_Posi;
	END_FOR
	iStep:=200;
	tDelay(IN:=FALSE , PT:=t#100ms , Q=> , ET=> );
200:
	bAxisNotMoving:=TRUE;
	FOR i:=MinHomeAxis TO MaxHomeAxis DO
		Axis_Interface[i].bMoveAbs:=FALSE ;
		bAxisNotMoving:=bAxisNotMoving AND AxisArr[i].Status.NotMoving;
	END_FOR
	tDelay(IN:=TRUE , PT:=t#100ms , Q=> , ET=> );
	IF bAxisNotMoving AND tDelay.Q  THEN
		iStep:=300;
	END_IF
300:
	All_Homed_OK:=TRUE;
	iStep:=0;
END_CASE
END_PROGRAM

(* POU 03_机台/05_HMI/PRG_AutoPreparation, ST *)
PROGRAM PRG_AutoPreparation
VAR
	iAutoHomeStep: INT;
	i: INT;
	iClearHomeStep: INT;
	bClearHome	:BOOL;(*清除回原信号*)
	rTrig:R_TRIG;
	bAxisNotMoving: BOOL;
	tDelay:TON;
END_VAR
rTrig(CLK:=bGoPrepareAuto OR bGoPrepareAuto_Cmd , Q=> );

CASE iAutoHomeStep OF
0:
	IF rTrig.Q AND All_Homed_OK THEN
		iAutoHomeStep:=50;
		bAutoReady:=FALSE;
	END_IF
50:
	FOR i:=1 TO NumOfCylinders DO
		stCtrlCylinder[i].bBack:=TRUE;	(*气缸回原*)
	END_FOR
	IF bAllCylinderBase THEN
		iAutoHomeStep:=100;
	END_IF
100:
	FOR i:=MinHomeAxis TO MaxHomeAxis DO
		stAxisParam[i].iTargetNr:=0;
		stHmiAxisCmd[i].bMoveAbs:=FALSE;
		Axis_Interface[i].fVelocity_of_Abs:=stAxisParam[i].fVelo_of_Posi;
	END_FOR
	iAutoHomeStep:=200;
200:
	FOR i:=MinHomeAxis TO MaxHomeAxis DO
		stHmiAxisCmd[i].bMoveAbs:=TRUE;
	END_FOR
	iAutoHomeStep:=300;
	tDelay(IN:=FALSE , PT:=t#20ms , Q=> , ET=> );
300:
	tDelay(IN:=TRUE , PT:=t#20ms , Q=> , ET=> );
	bAxisNotMoving:=TRUE;
	FOR i:=MinHomeAxis TO MaxHomeAxis DO
		Axis_Interface[i].bMoveAbs:=FALSE ;
		bAxisNotMoving:=bAxisNotMoving AND AxisArr[i].Status.NotMoving;
	END_FOR
	IF bAxisNotMoving AND tDelay.Q  THEN
		iAutoHomeStep:=400;
	END_IF
400:
	tDelay(IN:=FALSE , PT:=t#20ms , Q=> , ET=> );
	bAutoReady:=TRUE;
	iAutoHomeStep:=0;
END_CASE
END_PROGRAM

(* POU 02_Common/PRG_Estop, ST *)
PROGRAM PRG_Estop
VAR
	i: UINT;
END_VAR
FOR i:=MinHomeAxis TO MaxHomeAxis DO
(*使能*)
	(*IF i<>LEFTROLLER AND i<>RIGHTROLLER AND i<>Drive THEN		*)
		Axis_Interface[i].bEnable:=FALSE;		(*断开使能信号*)
		Axis_Interface[i].bEnableFw:=FALSE;
		Axis_Interface[i].bEnableBw:=FALSE;
		Axis_Interface[i].bHome:=FALSE;			(*由于急停时，张力还要有序放下，所以折3个轴应当有序断开*)
		Axis_Interface[i].bJog_Bw:=FALSE;
		Axis_Interface[i].bHalt:=FALSE;
		Axis_Interface[i].bJog_Fw:=FALSE;
		Axis_Interface[i].bMoveAbs:=FALSE;		(*张力轴如果断使能，会使得再次开机时立刻弹出，使得线松*)
		Axis_Interface[i].bMoveVelo:=FALSE;
		Axis_Interface[i].bMoveRel:=FALSE;
		Axis_Interface[i].bReset:=FALSE;
		Axis_Interface[i].bStop:=FALSE;
		Axis_Interface[i].bSetPos:=FALSE;
	(*END_IF*)
(*其他操作指令*)

END_FOR
END_PROGRAM

(* POU 03_机台/PRG_M_Function, ST *)
PROGRAM PRG_M_Function
VAR
	bGearIn_ZM	:	BOOL;
	bGearOut_ZM	:	BOOL;


END_VAR
(*气缸*)
PRG_Cylinder();
END_PROGRAM

(* POU 03_机台/04_气路/PRG_Cylinder, ST *)
PROGRAM PRG_Cylinder
VAR
	i:UINT;
END_VAR
FOR i:=1 TO NumOfCylinders DO


	stCtrlCylinder[i].fTimeOfContinue:=0.3;
	stCtrlCylinder[i].fTimeOfOvertime:=2;
	stCtrlCylinder[i].bContinue:=FALSE;


	fbCylinder[i](
		bContinue:=stCtrlCylinder[i].bContinue ,
		tContinueTime:= stCtrlCylinder[i].fTimeOfContinue ,
		tAlarmDelay:= stCtrlCylinder[i].fTimeOfOvertime ,
		DiWorkSensor:= stCtrlCylinder[i].DiWorkLimit ,
		DiBaseSensor:= stCtrlCylinder[i].DiBaseLimit ,
		Act:= stCtrlCylinder[i].bAct ,
		Back:= stCtrlCylinder[i].bBack ,
		Switch:= stCtrlCylinder[i].bSwitch ,
		AtAlarm=> stCtrlCylinder[i].CylinderAlarm_TimeOut,
		AtBasePos=>stCtrlCylinder[i].Cylinder_Limit_Base ,
		AtWorkPos=>stCtrlCylinder[i].Cylinder_Limit_Work,
		DoWorkPos=> stCtrlCylinder[i].DoAct,
		DoBasePos=> stCtrlCylinder[i].DoBack);
END_FOR

(***************************** 所有气缸都在原位的判断   ********************************************)
bAllCylinderBase:=TRUE;
FOR i:=1 TO NumOfCylinders DO
		bAllCylinderBase:=bAllCylinderBase AND stCtrlCylinder[i].Cylinder_Limit_Base;
END_FOR
END_PROGRAM

(* POU 02_Common/PRG_PTP, ST *)
PROGRAM PRG_PTP
VAR
	i: UINT;
	tCycleRead	:TON;

	SetRobotZ_Limit_Pos			 : ADSWRITE;
	SetRobotZ_Limit_Neg		 	: ADSWRITE;
	GetRobotZ_Limit_PosActive	: ADSWRITE;
	GetRobotZ_Limit_NegActive	: ADSWRITE;
	GetRobotZ_Limit_Pos			 : ADSWRITE;
	GetRobotZ_Limit_Neg		 	: ADSWRITE;


	tonWriteAds_Delay: TON;
	LastTorque: INT;

	bActive_PosLimit_GetRobot_Z: BOOL;
	bActive_NegLimit_GetRobot_Z: BOOL;
	bActive_PosLimit_GetRobot_Z_Old: BOOL;
	bActive_NegLimit_GetRobot_Z_Old: BOOL;
	bInit: BOOL;
	iStep: UINT;
	fbSoftLimit_Pos: ARRAY[1..5] OF ADSREAD;
	fbSoftLimit_Neg: ARRAY[1..5] OF ADSREAD;

	fbSoftLimit_Pos_w: ARRAY[1..5] OF ADSWRITE;
	fbSoftLimit_Neg_w: ARRAY[1..5] OF ADSWRITE;

	bNotBusy: BOOL;
	j,jj,jjj:UINT;

END_VAR
tCycleRead(IN:=NOT tCycleRead.Q , PT:=t#1s , Q=> , ET=> );

Act_AxisLimit();

FOR i:=1 TO MaxAxes DO
(*周期更新轴的数据*)
	axisarr[i].ReadStatus;

(*功能块调用*)
	aMC_Power[i](
		Enable:=Axis_Interface[i].bEnable ,
		Enable_Positive:=Axis_Interface[i].bEnableFw (*AND  NOT bSysEstop*) ,	(*放卷轴可能会因为正反向使能被锁定无法动弹反而无法完成急停后的松开动作*)
		Enable_Negative:=Axis_Interface[i].bEnableBw (*AND  NOT bSysEstop*),
		Override:=Axis_Interface[i].fOverride ,
		Axis:=axisarr[i],
		Status=>Axis_Interface[i].Axis_Ready );

	aMC_SetPos[i](
		Execute:=Axis_Interface[i].bSetPos AND NOT axisarr[i].Status.Coupled ,
		Position:=Axis_Interface[i].fPosition_ToBeSet ,
		Axis:=AxisArr[i]);

	aMC_Stop[i](
		Execute:=Axis_Interface[i].bStop AND NOT axisarr[i].Status.Coupled,
		Axis:=AxisArr[i]  );

	aMC_Reset[i](
		Execute:=(Axis_Interface[i].bReset OR bSysReset) AND AxisArr[i].Status.Error AND NOT axisarr[i].Status.Coupled,
		Axis:= AxisArr[i] );

	aMC_SoeReset[i](
		Execute:=(Axis_Interface[i].bReset OR bSysReset) AND AxisArr[i].Status.Error (*AND NOT axisarr[i].Status.Coupled*),
		Axis:=AxisArr[i] );

	aMC_Halt[i](
		Execute:=Axis_Interface[i].bHalt AND NOT axisarr[i].Status.Coupled ,
		Axis:= AxisArr[i] );

	aMC_Jog[i](
			JogForward:=Axis_Interface[i].bJog_Fw,
			JogBackwards:=Axis_Interface[i].bJog_Bw  ,
			Mode:=MC_JOGMODE_CONTINOUS ,
			Velocity:=Axis_Interface[i].fVelocity_of_Jog ,
			Axis:=axisarr[i]);

	aMC_MoveRelative[i]	(
		Execute:=Axis_Interface[i].bMoveRel ,
		Distance:=Axis_Interface[i].fPosition_of_Rel ,
		Velocity:=Axis_Interface[i].fVelocity_of_Rel ,
		Axis:=axisarr[i]);

	aMC_MoveAbsolute[i](
		Execute:=Axis_Interface[i].bMoveAbs ,
		Position:=Axis_Interface[i].fPositon_of_Abs ,
		Velocity:=Axis_Interface[i].fVelocity_of_Abs ,
		Axis:=axisarr[i]);

	aMC_MoveVelocity[i](
		Execute:=Axis_Interface[i].bMoveVelo ,
		Velocity:=Axis_Interface[i].fVelocity_of_Velo ,
		Direction:=MC_Negative_Direction ,
		Axis:=axisarr[i],
		InVelocity=>Axis_Interface[i].bInVelo);
END_FOR

(*状态的刷新以及综合状态的获取*)

All_Enable_OK:=TRUE;
AllAxesStandStill:=TRUE;
Axis_Has_error:=FALSE;
Axis_Homing:=FALSE;

FOR i:=1 TO MaxAxes DO
	All_Enable_OK:=All_Enable_OK AND AxisArr[i].Status.ControlLoopClosed;
	AllAxesStandStill:=AllAxesStandStill AND AxisArr[i].Status.NotMoving;
	Axis_Has_error:=Axis_Has_error OR AxisArr[i].Status.Error;
	Axis_Homing:=Axis_Homing OR AxisArr[i].Status.HomingBusy(*aMC_Home[i].Busy*);
	Axis_Interface[i].Axis_Homed:=AxisArr[i].Status.Homed;
	Axis_Interface[i].Axis_Err:=AxisArr[i].Status.Error;
	Axis_Interface[i].Axis_Coupled:= AxisArr[i].Status.Coupled;
	Axis_Interface[i].Axis_NotMoving:=AxisArr[i].Status.NotMoving;
	Axis_Interface[i].fActPos:=AxisArr[i].NcToPlc.ActPos;
	IF Axis_Interface[i].fActPos>0 THEN
		Axis_Interface[i].fActPosModbus:=REAL_TO_WORD(Axis_Interface[i].fActPos*10);
	ELSE
		Axis_Interface[i].fActPosModbus:=0;
	END_IF
	Axis_Interface[i].Axis_ErrID:=AxisArr[i].Status.ErrorID;
	stAxisDisplay[i].fActPos:=AxisArr[i].NcToPlc.ActPos;
	Axis_Interface[i].fActVelo:=AxisArr[i].NcToPlc.ActVelo;
	IF NOT (*aMC_Home[i].Busy*)AxisArr[i].Status.HomingBusy  THEN		(*使用轴本身的状态，而不是用具体的功能块更好*)	(*使用轴本身的状态优先级太低，轴先被使能信号停掉了，导致无法完成回零*)
		Axis_Interface[i].bEnableFw:=NOT Axis_Interface[i].Axis_Limit_Pos;
		Axis_Interface[i].bEnableBw:=NOT Axis_Interface[i].Axis_Limit_Neg;
	END_IF
END_FOR

Modbus_TCP;
Act_SoftLimitInit;
END_PROGRAM
ACTION Act_AxisLimit:
(*	1	顶部探头左
	2	顶部探头右	
	3	横向探头右	
	4	升降电机	
	5	准直电机	
	6	旋转电机	
	7	导轨电机	
	8	横向探头左	*)



FOR i:=1 TO 5 DO
IF iAxisSoftLimitSwitch_Pos[i]<>iAxisSoftLimitSwitch_Pos_Old[i] AND bInit THEN
	iAxisSoftLimitSwitch_Pos_Old[i]:=iAxisSoftLimitSwitch_Pos[i];
	fbSoftLimit_Pos_w[i].WRITE:=TRUE;
ELSE
	fbSoftLimit_Pos_w[i].WRITE:=FALSE;
END_IF

IF iAxisSoftLimitSwitch_Neg[i]<>iAxisSoftLimitSwitch_Neg_Old[i] AND bInit AND NOT fbSoftLimit_Pos_w[i].BUSY THEN
	iAxisSoftLimitSwitch_Neg_Old[i]:=iAxisSoftLimitSwitch_Neg[i];
	fbSoftLimit_Neg_w[i].WRITE:=TRUE;
ELSE
	fbSoftLimit_Neg_w[i].WRITE:=FALSE;
END_IF

IF  iAxisSoftLimitSwitch_Pos[i] THEN
	iAxisSoftLimitSwitch_Pos1[i]:=1;
ELSE
	iAxisSoftLimitSwitch_Pos1[i]:=0;
END_IF

IF  iAxisSoftLimitSwitch_Neg[i] THEN
	iAxisSoftLimitSwitch_Neg1[i]:=1;
ELSE
	iAxisSoftLimitSwitch_Neg1[i]:=0;
END_IF


END_FOR


FOR i:=1 TO 5 DO
fbSoftLimit_Pos_w[i](
	NETID:= '',
	PORT:=501 ,
	IDXGRP:=16#5000+i ,
	IDXOFFS:=16#C ,
	LEN:=2 ,
	SRCADDR:=ADR(iAxisSoftLimitSwitch_Pos1[i]) ,
	WRITE:= ,
	TMOUT:=t#200ms ,
	BUSY=> ,
	ERR=> , 
	ERRID=> );

fbSoftLimit_Neg_w[i](
	NETID:= '',
	PORT:=501 ,
	IDXGRP:=16#5000+i ,
	IDXOFFS:=16#B ,
	LEN:=2 ,
	SRCADDR:=ADR(iAxisSoftLimitSwitch_Neg1[i]) ,
	WRITE:= ,
	TMOUT:=t#200ms ,
	BUSY=> ,
	ERR=> , 
	ERRID=> );

END_FOR
END_ACTION
ACTION Act_SoftLimitinit:
(*	1	顶部探头左
	2	顶部探头右	
	3	横向探头右	
	4	升降电机	
	5	准直电机	
	6	旋转电机	
	7	导轨电机	
	8	横向探头左	*)

IF bInit THEN
	RETURN;
END_IF


CASE iStep OF
0:
	FOR i:=1 TO 5 DO
		fbSoftLimit_Pos[I].READ:=TRUE;
		fbSoftLimit_Neg[i].READ:=TRUE;
	END_FOR
	iStep:=100;
100:
	iStep:=200;

200:
	bNotBusy:=FALSE;
	FOR i:=1 TO 5 DO
		bNotBusy:=bNotBusy OR  fbSoftLimit_Pos[i].BUSY OR fbSoftLimit_Neg[i].BUSY;
	END_FOR
	IF NOT bNotBusy THEN
		iStep:=300;
	END_IF
300:
	FOR i:=1 TO 5 DO
		fbSoftLimit_Pos[I].READ:=FALSE;
		fbSoftLimit_Neg[i].READ:=FALSE;
	END_FOR
	iStep:=400;
400:
	bInit:=TRUE;
END_CASE



FOR i:=1 TO 5 DO
MEMSET(destAddr:=ADR(iAxisSoftLimitSwitch_Pos_Old[i]),fillByte:=0,n:=2);
MEMSET(destAddr:=ADR(iAxisSoftLimitSwitch_Neg_Old[i]),fillByte:=0,n:=2);
fbSoftLimit_Pos[i](
	NETID:='' ,
	PORT:= 501,
	IDXGRP:=16#5000+i ,
	IDXOFFS:=16#C ,
	LEN:=2 ,
	DESTADDR:=ADR(iAxisSoftLimitSwitch_Pos_Old[i]) ,
	READ:= , 
	TMOUT:=t#200ms ,
	BUSY=> , 
	ERR=> , 
	ERRID=> );

fbSoftLimit_Neg[i](
	NETID:='' ,
	PORT:= 501,
	IDXGRP:=16#5000+i ,
	IDXOFFS:=16#B ,
	LEN:=2 ,
	DESTADDR:=ADR(iAxisSoftLimitSwitch_Neg_Old[i]) ,
	READ:= , 
	TMOUT:=t#200ms ,
	BUSY=> , 
	ERR=> , 
	ERRID=> );


END_FOR
END_ACTION
ACTION Modbus_TCP:
(**************************************************	转运组X轴   read  	****************************************************************************)
mb_Output_Registers[1]	:=	BOOL_TO_WORD(Axis_Interface[1].Axis_Ready)	;	(*	X轴准备就绪	*)
mb_Output_Registers[2]	:=	BOOL_TO_WORD(Axis_Interface[1].Axis_Err)	;	(*	X轴报警	*)
mb_Output_Registers[3]	:=	BOOL_TO_WORD(NOT Axis_Interface[1].Axis_NotMoving)	;	(*	X轴运行中	*)
mb_Output_Registers[4]	:=	BOOL_TO_WORD(Axis_Interface[1].Axis_Limit_Pos)	;	(*	X轴正限位	*)
mb_Output_Registers[5]	:=	BOOL_TO_WORD(Axis_Interface[1].Axis_Limit_Neg)	;	(*	X轴负限位	*)
mb_Output_Registers[6]	:=	Axis_Interface[1].fActPosModbus	;	(*	X轴当前位置	*)
mb_Output_Registers[7]	:=	UDINT_TO_WORD(Axis_Interface[1].Axis_ErrID)	;	(*	X轴报警代码	*)
mb_Output_Registers[8]	:=	BOOL_TO_WORD(Axis_Interface[1].bEnable)	;	(*	X轴使能	*)

(**************************************************	转运组Z轴   read  	****************************************************************************)
mb_Output_Registers[9]	:=	BOOL_TO_WORD(Axis_Interface[2].Axis_Ready)	;	(*	z轴准备就绪	*)
mb_Output_Registers[10]	:=	BOOL_TO_WORD(Axis_Interface[2].Axis_Err)	;	(*	Z轴报警	*)
mb_Output_Registers[11]	:=	BOOL_TO_WORD(NOT Axis_Interface[2].Axis_NotMoving)	;	(*	Z轴运行中	*)
mb_Output_Registers[12]	:=	BOOL_TO_WORD(Axis_Interface[2].Axis_Limit_Pos)	;	(*	Z轴正限位	*)
mb_Output_Registers[13]	:=	BOOL_TO_WORD(Axis_Interface[2].Axis_Limit_Neg)	;	(*	X轴负限位	*)
mb_Output_Registers[14]	:=	Axis_Interface[2].fActPosModbus	;	(*	Z轴当前位置	*)
mb_Output_Registers[15]	:=	UDINT_TO_WORD(Axis_Interface[2].Axis_ErrID)	;	(*	Z轴报警代码	*)
mb_Output_Registers[16]	:=	BOOL_TO_WORD(Axis_Interface[2].bEnable)	;	(*	Z轴使能	*)

(**************************************************	裁剪模组X轴   read  	****************************************************************************)
mb_Output_Registers[17]	:=	BOOL_TO_WORD(Axis_Interface[3].Axis_Ready)	;	(*	X轴准备就绪	*)
mb_Output_Registers[18]	:=	BOOL_TO_WORD(Axis_Interface[3].Axis_Err)	;	(*	X轴报警	*)
mb_Output_Registers[19]	:=	BOOL_TO_WORD(NOT Axis_Interface[3].Axis_NotMoving)	;	(*	X轴运行中	*)
mb_Output_Registers[20]	:=	BOOL_TO_WORD(Axis_Interface[3].Axis_Limit_Pos)	;	(*	X轴正限位	*)
mb_Output_Registers[21]	:=	BOOL_TO_WORD(Axis_Interface[3].Axis_Limit_Neg)	;	(*	X轴负限位	*)
mb_Output_Registers[22]	:=	Axis_Interface[3].fActPosModbus	;	(*	X轴当前位置	*)
mb_Output_Registers[23]	:=	UDINT_TO_WORD(Axis_Interface[3].Axis_ErrID)	;	(*	X轴报警代码	*)
mb_Output_Registers[24]	:=	BOOL_TO_WORD(Axis_Interface[3].bEnable)	;	(*	X轴使能	*)

(**************************************************	裁剪模组Y轴   read  	****************************************************************************)
mb_Output_Registers[25]	:=	BOOL_TO_WORD(Axis_Interface[4].Axis_Ready)	;	(*	Y轴准备就绪	*)
mb_Output_Registers[26]	:=	BOOL_TO_WORD(Axis_Interface[4].Axis_Err)	;	(*	Y轴报警	*)
mb_Output_Registers[27]	:=	BOOL_TO_WORD(NOT Axis_Interface[4].Axis_NotMoving)	;	(*	Y轴运行中	*)
mb_Output_Registers[28]	:=	BOOL_TO_WORD(Axis_Interface[4].Axis_Limit_Pos)	;	(*	Y轴正限位	*)
mb_Output_Registers[29]	:=	BOOL_TO_WORD(Axis_Interface[4].Axis_Limit_Neg)	;	(*	Y轴负限位	*)
mb_Output_Registers[30]	:=	Axis_Interface[4].fActPosModbus	;	(*	Y轴当前位置	*)
mb_Output_Registers[31]	:=	UDINT_TO_WORD(Axis_Interface[4].Axis_ErrID)	;	(*	Y轴报警代码	*)
mb_Output_Registers[32]	:=	BOOL_TO_WORD(Axis_Interface[4].bEnable)	;	(*	Y轴使能	*)

(**************************************************	拧瓶盖轴   read  	****************************************************************************)
mb_Output_Registers[33]	:=	BOOL_TO_WORD(Axis_Interface[5].Axis_Ready)	;	(*	R轴准备就绪	*)
mb_Output_Registers[34]	:=	BOOL_TO_WORD(Axis_Interface[5].Axis_Err)	;	(*	R轴报警	*)
mb_Output_Registers[35]	:=	BOOL_TO_WORD(NOT Axis_Interface[5].Axis_NotMoving)	;	(*	R轴运行中	*)
mb_Output_Registers[36]	:=	BOOL_TO_WORD(Axis_Interface[5].Axis_Limit_Pos)	;	(*	R轴正限位	*)
mb_Output_Registers[37]	:=	BOOL_TO_WORD(Axis_Interface[5].Axis_Limit_Neg)	;	(*	R轴负限位	*)
mb_Output_Registers[38]	:=	Axis_Interface[5].fActPosModbus	;	(*	R轴当前位置	*)
mb_Output_Registers[39]	:=	UDINT_TO_WORD(Axis_Interface[5].Axis_ErrID)	;	(*	R轴报警代码	*)
mb_Output_Registers[40]	:=	BOOL_TO_WORD(Axis_Interface[5].bEnable)	;	(*	R轴使能	*)

(**************************************************	气缸   read  	****************************************************************************)
FOR j:=1 TO NumOfCylinders DO
	mb_Output_Registers[41+(j-1)*3]	:=	BOOL_TO_WORD(stCtrlCylinder[j].DoAct)	;	(*	气缸的工作输出	*)
	mb_Output_Registers[42+(j-1)*3]	:=	BOOL_TO_WORD(stCtrlCylinder[j].DiWorkLimit)	;	(*	气缸的正限位输入	*)
	mb_Output_Registers[43+(j-1)*3]	:=	BOOL_TO_WORD(stCtrlCylinder[j].DiBaseLimit)	;	(*	气缸的负限位输入	*)
END_FOR



(**************************************************	转运组X轴   write  	****************************************************************************)
stAxisParam[1].fTargetPosi		:= mb_Output_Registers[155]	;	(*转运组 X轴的目标位置*)
stAxisParam[1].WorkPos1		:= mb_Output_Registers[156]	;	(*转运组 X轴的工作位置1*)
stAxisParam[1].WorkPos2		:= mb_Output_Registers[157]	;	(*转运组 X轴的工作位置2*)
stAxisParam[1].WorkPos3		:= mb_Output_Registers[158]	;	(*转运组 X轴的工作位置3*)
iPos_X_Axis 					:= mb_Output_Registers[159	]	;	(*转运组X轴的目标位置运动命令*)
stHmiAxisCmd[1].bHome		:= WORD_TO_BOOL(mb_Output_Registers[160])	;	(*转运组X轴回原点设置命令*)
stHmiAxisCmd[1].bEnable		:= WORD_TO_BOOL(mb_Output_Registers[161])	;	(*转运组X轴使能设置命令*)
stHmiAxisCmd[1].bSetBiasBnt 	:=WORD_TO_BOOL( mb_Output_Registers[162])	;	(*转运组X轴原点设置命令*)
Axis_Interface[1].bStop			:= WORD_TO_BOOL(mb_Output_Registers[163])	;	(*转运组X轴停止设置命令*)
stHmiAxisCmd[1].bReset		:= WORD_TO_BOOL(mb_Output_Registers[164])	;	(*转运组X轴复位设置命令*)

(**************************************************	转运组Y轴   write  	****************************************************************************)
stAxisParam[2].fTargetPosi		:= mb_Output_Registers[165]	;	(*轴的目标位置*)
stAxisParam[2].WorkPos1		:= mb_Output_Registers[166]	;	(*轴的工作位置1*)
stAxisParam[2].WorkPos2		:= mb_Output_Registers[167]	;	(*轴的工作位置2*)
stAxisParam[2].WorkPos3		:= mb_Output_Registers[168]	;	(*轴的工作位置3*)
iPos_Z_Axis 					:= mb_Output_Registers[169	]	;	(*轴的目标位置运动命令*)
stHmiAxisCmd[2].bHome		:= WORD_TO_BOOL(mb_Output_Registers[170])	;	(*轴回原点设置命令*)
stHmiAxisCmd[2].bEnable		:= WORD_TO_BOOL(mb_Output_Registers[171])	;	(*轴使能设置命令*)
stHmiAxisCmd[2].bSetBiasBnt 	:=  WORD_TO_BOOL(mb_Output_Registers[172])	;	(*轴原点设置命令*)
Axis_Interface[2].bStop			:=  WORD_TO_BOOL(mb_Output_Registers[173])	;	(*轴停止设置命令*)
stHmiAxisCmd[2].bReset		:=  WORD_TO_BOOL(mb_Output_Registers[174])	;	(*轴复位设置命令*)

(**************************************************	裁剪模组X轴   write  	****************************************************************************)
stAxisParam[3].fTargetPosi		:= mb_Output_Registers[175]	;	(*轴的目标位置*)
stAxisParam[3].WorkPos1		:= mb_Output_Registers[176]	;	(*轴的工作位置1*)
stAxisParam[3].WorkPos2		:= mb_Output_Registers[177]	;	(*轴的工作位置2*)
stAxisParam[3].WorkPos3		:= mb_Output_Registers[178]	;	(*轴的工作位置3*)
iPos_X2_Axis 				:= mb_Output_Registers[179	]	;	(*轴的目标位置运动命令*)
stHmiAxisCmd[3].bHome		:=  WORD_TO_BOOL(mb_Output_Registers[180])	;	(*轴回原点设置命令*)
stHmiAxisCmd[3].bEnable		:=  WORD_TO_BOOL(mb_Output_Registers[181])	;	(*轴使能设置命令*)
stHmiAxisCmd[3].bSetBiasBnt 	:=  WORD_TO_BOOL(mb_Output_Registers[182])	;	(*轴原点设置命令*)
Axis_Interface[3].bStop			:=  WORD_TO_BOOL(mb_Output_Registers[183])	;	(*轴停止设置命令*)
stHmiAxisCmd[3].bReset		:=  WORD_TO_BOOL(mb_Output_Registers[184])	;	(*轴复位设置命令*)
(**************************************************	裁剪模组Y轴   write  	****************************************************************************)
stAxisParam[4].fTargetPosi		:= mb_Output_Registers[185]	;	(*轴的目标位置*)
stAxisParam[4].WorkPos1		:= mb_Output_Registers[186]	;	(*轴的工作位置1*)
stAxisParam[4].WorkPos2		:= mb_Output_Registers[187]	;	(*轴的工作位置2*)
stAxisParam[4].WorkPos3		:= mb_Output_Registers[188]	;	(*轴的工作位置3*)
iPos_Y2_Axis 				:= mb_Output_Registers[189	]	;	(*轴的目标位置运动命令*)
stHmiAxisCmd[4].bHome		:=  WORD_TO_BOOL(mb_Output_Registers[190])	;	(*轴回原点设置命令*)
stHmiAxisCmd[4].bEnable		:=  WORD_TO_BOOL(mb_Output_Registers[191])	;	(*轴使能设置命令*)
stHmiAxisCmd[4].bSetBiasBnt 	:=  WORD_TO_BOOL(mb_Output_Registers[192])	;	(*轴原点设置命令*)
Axis_Interface[4].bStop			:=  WORD_TO_BOOL(mb_Output_Registers[193])	;	(*轴停止设置命令*)
stHmiAxisCmd[4].bReset		:=  WORD_TO_BOOL(mb_Output_Registers[194])	;	(*轴复位设置命令*)

(**************************************************	旋转轴   write  	****************************************************************************)
stAxisParam[5].fTargetPosi		:= mb_Output_Registers[195]	;	(*轴的目标位置*)
stAxisParam[5].WorkPos1		:= mb_Output_Registers[196]	;	(*轴的工作位置1*)
stAxisParam[5].WorkPos2		:= mb_Output_Registers[197]	;	(*轴的工作位置2*)
stAxisParam[5].WorkPos3		:= mb_Output_Registers[198]	;	(*轴的工作位置3*)
iPos_R_Axis 					:= mb_Output_Registers[199	]	;	(*轴的目标位置运动命令*)
stHmiAxisCmd[5].bHome		:= WORD_TO_BOOL(mb_Output_Registers[200])	;	(*轴回原点设置命令*)
stHmiAxisCmd[5].bEnable		:= WORD_TO_BOOL(mb_Output_Registers[201])	;	(*轴使能设置命令*)
stHmiAxisCmd[5].bSetBiasBnt 	:= WORD_TO_BOOL(mb_Output_Registers[202])	;	(*轴原点设置命令*)
Axis_Interface[5].bStop			:= WORD_TO_BOOL(mb_Output_Registers[203])	;	(*轴停止设置命令*)
stHmiAxisCmd[5].bReset		:= WORD_TO_BOOL(mb_Output_Registers[204])	;	(*轴复位设置命令*)

(**************************************************	气缸   wirte 	****************************************************************************)
FOR jj:=1 TO NumOfCylinders DO
	stCtrlCylinder[j].DoAct := WORD_TO_BOOL(mb_Output_Registers[205+jj-1]);
END_FOR
iGoAutoTogether_Cmd		:=	mb_Output_Registers[243]		;	(*一键启动*)
iGoHomeTogether_Cmd	:=	mb_Output_Registers[244]		;	(*一键回原点*)
iGoResetTogether_Cmd	:=	mb_Output_Registers[245]		;	(*一键复位*)
iGoStopTogether_Cmd		:= 	mb_Output_Registers[246]		;	(*一键停止*)
iGoPrepareAuto_Cmd	:=	mb_Output_Registers[247]		;	(*一键去准备位*)
iAuto_Cmd	:=	mb_Output_Registers[248]		;	(*自动切换*)
END_ACTION

(* POU 06_自动/PRG_AutoWork, ST *)
PROGRAM PRG_AutoWork
VAR
	iGetPaperStep:UINT;
	riGetPaper_Cmd:R_TRIG;

	iCollectStep:UINT;
	riCollect_Cmd:R_TRIG;

	iPutStep:UINT;
	riPut_Cmd:R_TRIG;

	iCutStep:UINT;
	riCut_Cmd:R_TRIG;


	iSetBoxStep:UINT;
	riSetBox_Cmd:R_TRIG;



	tDelay:TON;


END_VAR
;
END_PROGRAM
ACTION Act_Collect:
riCollect_Cmd(CLK:=bCollect_Cmd , Q=> );
CASE iCollectStep OF
	0:
		IF riCollect_Cmd.Q AND bHasGot_Paper THEN
			iCollectStep:=10;
			bHasCollected:=FALSE;
		END_IF
	10:
		stCtrlCylinder[1].bAct:=TRUE;		(*采集组?采集盖下压气缸1工作位*)
		stCtrlCylinder[2].bAct:=TRUE;		(*采集组?采集盖下压气缸2工作位*)
		IF stCtrlCylinder[1].Cylinder_Limit_Work AND stCtrlCylinder[2].Cylinder_Limit_Work THEN		(*检测到已经到位*)
			iCollectStep:=20;
		END_IF

	20:
		tDelay(IN:=TRUE , PT:=t#10000ms , Q=> , ET=> );
		IF tDelay.Q THEN
			iCollectStep:=30;
		END_IF
	30:
		stCtrlCylinder[1].bBack:=TRUE;		(*采集组?采集盖下压气缸1回基位*)
		stCtrlCylinder[2].bBack:=TRUE;		(*采集组?采集盖下压气缸2回基位*)
		IF stCtrlCylinder[1].Cylinder_Limit_Base AND stCtrlCylinder[2].Cylinder_Limit_Base THEN		(*检测到已经到位*)
			iCollectStep:=0;
			bHasCollected:=TRUE;
		END_IF
END_ACTION
ACTION Act_GetPaper:
riGetPaper_Cmd(CLK:=bGet_Paper_Cmd , Q=> );
CASE iGetPaperStep OF
	0:
		IF riGetPaper_Cmd.Q THEN
			iGetPaperStep:=5;
			bHasGot_Paper:=FALSE;
		END_IF

	5:
		IF ABS(Axis_Interface[1].fPositon_of_Abs)<0.1 THEN	(*转运模组X轴起始位保持*)
			iGetPaperStep:=10;
		ELSE
			Axis_Interface[1].fPositon_of_Abs:= 0;
		END_IF

	10:
		IF ABS(Axis_Interface[2].fPositon_of_Abs - stAxisParam[2].WorkPos1)<0.1 THEN	(*转运模组Z轴到工位1准备取滤纸*)
			iGetPaperStep:=20;
		ELSE
			Axis_Interface[2].fPositon_of_Abs := stAxisParam[2].WorkPos1;
		END_IF

	20:
		stCtrlCylinder[3].bAct:=TRUE;		(*滤纸转运组吸盘气缸工作位*)
		IF stCtrlCylinder[3].Cylinder_Limit_Work THEN		(*检测到已经到位*)
			iGetPaperStep:=30;
		END_IF
	30:
		IF ABS(Axis_Interface[2].fPositon_of_Abs - stAxisParam[2].WorkPos2)<0.1 THEN	(*转运模组Z轴到工位2转运位*)
			iGetPaperStep:=40;
		ELSE
			Axis_Interface[2].fPositon_of_Abs := stAxisParam[2].WorkPos2;
		END_IF

	40:
		IF ABS(Axis_Interface[1].fPositon_of_Abs - stAxisParam[1].WorkPos1)<0.1 THEN	(*转运模组X轴到工位1*)
			iGetPaperStep:=50;
		ELSE
			Axis_Interface[1].fPositon_of_Abs := stAxisParam[1].WorkPos1;
		END_IF

	50:
		IF ABS(Axis_Interface[2].fPositon_of_Abs - stAxisParam[2].WorkPos3)<0.1 THEN	(*转运模组Z轴到工位3采集组滤纸下放位*)
			iGetPaperStep:=60;
		ELSE
			Axis_Interface[2].fPositon_of_Abs := stAxisParam[2].WorkPos3;
		END_IF

	60:
		stCtrlCylinder[3].bBack:=FALSE;		(*滤纸转运组吸盘气缸回基位*)
		IF stCtrlCylinder[3].Cylinder_Limit_Base THEN		(*检测到已经到位*)
			iGetPaperStep:=70;
		END_IF

	70:
		IF ABS(Axis_Interface[2].fPositon_of_Abs - stAxisParam[2].WorkPos2)<0.1 THEN	(*转运模组Z轴到工位2下放后回到转运位*)
			iGetPaperStep:=80;
		ELSE
			Axis_Interface[2].fPositon_of_Abs := stAxisParam[2].WorkPos2;
		END_IF

	80:
		IF ABS(Axis_Interface[1].fPositon_of_Abs)<0.1 THEN	(*转运模组X轴回起始位保持*)
			bHasGot_Paper:=TRUE;
			iGetPaperStep:=0;
		ELSE
			Axis_Interface[1].fPositon_of_Abs:= 0;
		END_IF

	END_CASE
END_ACTION

(* POU 03_机台/04_气路/FB_Cylinder, ST *)
FUNCTION_BLOCK FB_Cylinder
VAR_INPUT
(*PLC parameter*)
	bContinue			:BOOL:=FALSE;		(*true为连续动作*)
	tContinueTime		:REAL:=1;	(*单位秒，从动作开始记时，达到这个时间回退*)
	tAlarmDelay			:REAL:=1;	(*单位秒，长时间没有达到预定动作报警*)
(*From DI*)
	DiWorkSensor		:BOOL;	(*动作时触发的传感器*)
	DiBaseSensor		:BOOL;	(*初始位置触发的传感器*)
END_VAR
VAR_OUTPUT
(*To PLC*)
	AtAlarm			:BOOL;	(*报警，多气缸联动报警在自动程序里做，不要做在单气缸里面*)(*报警信号输出一个周期的脉冲信号*)
	AtBasePos		:BOOL;		(*在初始位*)
	AtWorkPos		:BOOL;		(*在工作位*)
(*To DO*)
	DoWorkPos		:BOOL;	(*输出给气缸，true使之动作*)
	DoBasePos		:BOOL;	(*输出给气缸，可以悬空*)
END_VAR
VAR_IN_OUT
(*PLC command*)
	Act					:BOOL;	(*动作，程序使用*)
	Back				:BOOL;	(*回位，程序使用*)
	Switch				:BOOL;	(*切换状态，程序使用*)
END_VAR
VAR
	tonAlarm,tonContinue		:TON;
	iStep						: UINT;
	fTrigWork,fTrigBase,fTrigSwitch	:R_TRIG;	(*1125改为上升沿了*)
	AlarmDelay					:TON;
	tonAct,tonBack				:TON;
	tLastCmd					:TIME:=t#100ms;
END_VAR
fTrigWork(CLK:= Act, Q=> );
fTrigBase(CLK:=Back, Q=> );
fTrigSwitch(CLK:=Switch , Q=> );

tonAct(IN:=Act , PT:=tLastCmd , Q=> , ET=> );
tonBack(IN:=Back , PT:=tLastCmd , Q=> , ET=> );

IF tonAct.Q THEN Act:=FALSE;END_IF
IF tonBack.Q THEN Back:=FALSE;END_IF

(*******切换状态 ********)
IF fTrigSwitch.Q AND iStep=0  THEN
	Switch:=FALSE;
	IF DiWorkSensor OR DoWorkPos THEN iStep:=200;
	ELSIF DiBaseSensor OR DoBasePos  THEN iStep:=100;
	END_IF
ELSIF iStep<>0 THEN
	Switch:=FALSE;
END_IF

(*两个输出取反*)
DoBasePos:=NOT DoWorkPos;

CASE iStep OF
0:
	AtAlarm:=FALSE;
	tonAlarm(IN:=FALSE);
	tonContinue(IN:=FALSE);
	IF fTrigWork.Q AND NOT bContinue  THEN
		iStep:=100;
	ELSIF fTrigWork.Q AND bContinue THEN
		iStep:=150;
	ELSIF fTrigBase.Q THEN
		iStep:=200;
	END_IF
	tonAlarm(IN:=FALSE);
100:
	DoWorkPos:=TRUE;
	tonAlarm(IN:=TRUE , PT:=REAL_TO_TIME(tAlarmDelay*1000) , Q=> , ET=> );
	AlarmDelay(in:=FALSE);
	IF DiWorkSensor AND NOT DiBaseSensor  THEN
		iStep:=0;
	ELSIF tonAlarm.Q THEN
		AtAlarm:=TRUE;
		iStep:=990;
	END_IF
150:
	DoWorkPos:=TRUE;
	tonContinue(IN:=TRUE , PT:=REAL_TO_TIME(tContinueTime*1000) , Q=> , ET=> );
	IF tonContinue.Q THEN
		tonContinue(IN:=FALSE);
		iStep:=200;
	END_IF
200:
	DoWorkPos:=FALSE;
	tonAlarm(IN:=TRUE , PT:=REAL_TO_TIME(tAlarmDelay*1000) , Q=> , ET=> );
	IF NOT DiWorkSensor AND  DiBaseSensor  THEN
		iStep:=0;
	ELSIF tonAlarm.Q THEN
		AtAlarm:=TRUE;
		iStep:=990;
	END_IF
990:
	AlarmDelay(in:=TRUE,pt:=t#0.1s);
	IF  AlarmDelay.Q THEN
		iStep:=0;
	END_IF
END_CASE


(***************************  状态判定  *****************************)
IF   DiBaseSensor AND NOT DiWorkSensor  THEN
	AtWorkPos:=FALSE;
	AtBasePos:=TRUE;
ELSIF NOT DiBaseSensor AND DiWorkSensor THEN
	AtWorkPos:=TRUE;
	AtBasePos:=FALSE;
ELSIF NOT DiBaseSensor AND NOT DiWorkSensor THEN
	AtWorkPos:=FALSE;
	AtBasePos:=FALSE;
END_IF
END_FUNCTION_BLOCK

(* POU 00_Basic/PulseGenerator/PulseCtrl, ST *)
FUNCTION_BLOCK PulseCtrl
VAR_INPUT
END_VAR
VAR_OUTPUT
	BlinkSlow		: BOOL;
	Blink				: BOOL;
	BlinkFast		: BOOL;
	BlinkVeryFast	:	BOOL;
END_VAR
VAR
	_20ms			: PulseGeneratorCtrl;
	_100ms			: PulseGeneratorCtrl;
	_250ms			: PulseGeneratorCtrl;
	_400ms			: PulseGeneratorCtrl; (* Blink Fast *)
	_500ms			: PulseGeneratorCtrl;
	_800ms			: PulseGeneratorCtrl; (* Blink *)
	_1s				: PulseGeneratorCtrl;
	_1s600ms			: PulseGeneratorCtrl; (* Blink Slow *)
(*	_2s				: PulseGeneratorCtrl; *)
	_5s				: PulseGeneratorCtrl;
(*	_10s				: PulseGeneratorCtrl; *)
(*	_2m				: PulseGeneratorCtrl; *)
(*	_5m				: PulseGeneratorCtrl; *)
(*	_30m				: PulseGeneratorCtrl; *)
END_VAR
(* Taktgeber *******************************************************************************)
	(* Generiere 100ms Takt *)
	_20ms(
		PT_OFF			:= t#20ms,
		PT_ON				:= t#20ms,
		Q					=> ,
		RT					=> );

	(* Generiere 100ms Q *)
	_100ms(
		PT_OFF			:= t#100ms,
		PT_ON				:= t#100ms,
		Q					=> ,
		RT					=> );

	(* Generiere 250ms Q Flimmerlicht*)
	_250ms(
		PT_OFF			:= t#250ms,
		PT_ON				:= t#250ms,
		Q					=> BlinkVeryFast,
		RT					=> );

	(* Generiere 400ms Q Schnelles Blinklicht *)
	_400ms(
		PT_OFF			:= t#400ms,
		PT_ON				:= t#400ms,
		Q					=> BlinkFast,
		RT					=> ); 

	(* Generiere 500ms Q *)
	_500ms(
		PT_OFF			:= t#500ms,
		PT_ON				:= t#500ms,
		Q					=> ,
		RT					=> );

	(* Generiere 800ms Q Blinklicht *)
	_800ms(
		PT_OFF			:= t#800ms,
		PT_ON				:= t#800ms,
		Q					=> Blink, 
		RT					=> );

	(* Generiere 1s Q *)
	_1s(
		PT_OFF			:= t#1s,
		PT_ON				:= t#1s,
		Q					=> ,
		RT					=> );

	(* Generiere 1s600ms Q Langsames Blinklicht *)
	_1s600ms(
		PT_OFF			:= t#1s600ms,
		PT_ON				:= t#1s600ms,
		Q					=> BlinkSlow,
		RT					=> );

	(* Generiere 2s Q *)
(*	_2s(
		PT_OFF			:= t#2s,
		PT_ON				:= t#2s,
		Q					=> ,
		RT					=> ); *)

	(* Generiere 2s Q *)
	_5s(
		PT_OFF			:= t#5s,
		PT_ON				:= t#5s,
		Q					=> ,
		RT					=> );

	(* Generiere 10s Q *)
(*	_10s(
		PT_OFF			:= t#10s,
		PT_ON				:= t#10s,
		Q					=> ,
		RT					=> ); *)

	(* Generiere 2Min Q *)
(*	_2m(
		PT_OFF			:= t#2m,
		PT_ON				:= t#2m,
		Q					=> ,
		RT					=> ); *)

	(* Generiere 5Min Q *)
(*	_5m(
		PT_OFF			:= t#5m,
		PT_ON				:= t#5m,
		Q					=> ,
		RT					=> ); *)

	(* Generiere 30Min Q *)
(*	_30m(
		PT_OFF			:= t#30m,
		PT_ON				:= t#30m,
		Q					=> ,
		RT					=> ); *)

(************************************************************************************************)
END_FUNCTION_BLOCK

(* POU 00_Basic/PulseGenerator/PulseGeneratorCtrl, ST *)
FUNCTION_BLOCK PulseGeneratorCtrl
VAR_INPUT
	PT_OFF		: TIME;
	PT_ON			: TIME;
END_VAR
VAR_OUTPUT
	Q				: BOOL;
	RT				: BOOL;
END_VAR
VAR
	TON_PULSE		: TON;
END_VAR
(* Reset Flanke *)
RT := FALSE;
(* Taktgenerator *)
IF TON_PULSE.Q AND Q THEN
	TON_PULSE(IN:=FALSE  , PT:= PT_OFF);
	RT := Q;
	Q := FALSE;
ELSIF	TON_PULSE.Q AND NOT Q THEN
	RT := NOT Q;
	TON_PULSE(IN:= FALSE , PT:= PT_ON) ;
	Q := TRUE;
END_IF
(* Work Timer *)
TON_PULSE(IN:=TRUE);

(*************************************************************)
END_FUNCTION_BLOCK

(* POU 00_Basic/SystemInfo/SystemInfoCtrl, ST *)
FUNCTION_BLOCK SystemInfoCtrl
VAR_INPUT
	Reset					: BOOL;
	RTCSyncCylce		:	DWORD := 5; (* in seconds *)
	TimeStampTrig		:	BOOL;
END_VAR
VAR_OUTPUT
	RunTimeNo			: BYTE;
	ProjectName			: STRING(32);
	NumberOfTasks		: BYTE;
	OnlineChangeCount	: UINT;
	RetainVarErr		: BOOL;
	PersistenVarErr	: BOOL;
	TimeStampDT			:	DATE_AND_TIME;
	TimeStamp			:	STRING(25); (* DD.MM.YY-Stunde:Minute:Sekunde:xxx *)
	TimeStr				:	STRING(15);	(* hh.mm.ss.xxms *)
	DateStr				:	STRING(15);	(* dd.mm.jj *)
	TimeStamp2			:	STRING(25); (* YYYY-MM-DD_HHMMSS for example YYYY-MM-DD_HHMMSS_Name.txt *)
	TimeStruct			:	TIMESTRUCT;
	MonthDays			:	WORD;
	LeapYear				:	BOOL;
	WeekOfYear			:	WORD;
	timezoneId			: 	E_TimeZoneID;
END_VAR

VAR
	(* Inst. Get Taskindex *)
	InstGETCURTASKINDEX	: 	GETCURTASKINDEX;
	InstLocalSystemTime	:	FB_LocalSystemTime;

	(* Info: SystemInfo.bootDataFlags
	Bit
	0 RETAIN Variablen: LOADED (fehlerfrei geladen)
	1 RETAIN Variablen: INVALID (es wurde die Sicherungskopie geladen, weil keine gültige Datei vorhanden war)
	2 RETAIN Variablen: REQUESTED (RETAIN Variablen sollten geladen werden, Einstellung im TwinCAT System Control))
	3 reserviert
	4 PERSISTENT Variablen: LOADED (fehlerfrei geladen)
	5 PERSISTENT Variablen: INVALID (es wurde die Sicherungskopie geladen, weil keine gültige Datei vorhanden war)
	6 reserviert
	7 reserviert *)

	RetainVarLoaded			: BOOL;
	RetainVarInvalid		: BOOL;
	RetainVarRequested		: BOOL;
	PersistentVarLoaded		: BOOL;
	PersistentVarInvalid	: BOOL;

	(* Info: SystemTaskInfoArr	(* Ist ein Array von 1-4 *)
	active					:	BOOL; 		(* Diese Variable zeigt an, ob die Task aktiv ist.*)
	taskName					:	STRING(16);	(* Der Taskname.*)
	firstCycle				:	BOOL;			(* Diese Variable hat im ersten Zyklus der SPS-Task den Wert: TRUE.*)
	cycleTimeExceeded		:	BOOL;			(* In dieser Variablen wird ein 躡erschreiten der eingestellten Taskzykluszeit gemeldet*)
	cycleTime				:	UDINT;		(* Eingestellte Taskzykluszeit in Vielfachen von 100ns*)
	lastExecTime			:	UDINT;		(* Benötigte Zykluszeit für den letzten Zyklus in Vielfachen von 100 ns*)
	priority					:	BYTE;			(* Eingestellte Prioritaet der Task*)
	cycleCount				: 	UDINT;		(* Zykluszaehler*) *)
	_sec						:	WORD;
	_hour						:	WORD;
END_VAR
(* Get Current Task Index ************************************************************************)
	InstGETCURTASKINDEX();

(* Read System Info Current Task *****************************************************************)
	(* Task Info *)
	RunTimeNo				:= SystemInfo.runTimeNo;
	ProjectName				:= SystemInfo.projectName;
	NumberOfTasks 			:= SystemInfo.numberOfTasks;
	OnlineChangeCount		:= SystemInfo.onlineChangeCount;

	(* System Boot Flags *)
	RetainVarLoaded		:= SystemInfo.bootDataFlags.0;
	RetainVarInvalid		:= SystemInfo.bootDataFlags.1 ;
	RetainVarRequested 	:= SystemInfo.bootDataFlags.2 ;
	PersistentVarLoaded	:= SystemInfo.bootDataFlags.4;
	PersistentVarInvalid	:= SystemInfo.bootDataFlags.5;


	(* Retein/Persisten Data Err *)
	IF SystemTaskInfoArr[InstGETCURTASKINDEX.Index].firstCycle THEN
		RetainVarErr		:= NOT RetainVarLoaded AND RetainVarRequested OR RetainVarInvalid;
		PersistenVarErr	:= NOT PersistentVarLoaded OR PersistentVarInvalid;
	ELSIF Reset THEN
		M_Reset();
	ELSE
		;
	END_IF

(* Systemzeit auslesen ************************************************************************)
	InstLocalSystemTime(
		sNetID		:= '',
		bEnable		:= TRUE,
		dwCycle		:= RTCSyncCylce,
		dwOpt			:= (* Default *),
		tTimeout		:= (* Default *),
		bValid		=> ,
		systemTime	=> TimeStruct,
		tzID			=> timezoneId);

	IF TimeStampTrig
		AND InstLocalSystemTime.bValid
	THEN
		(* Date dd.mm.jj ********************)
		IF TimeStruct.wDay < 10 THEN
			DateStr := CONCAT('0',WORD_TO_STRING(TimeStruct.wDay));
		ELSE
			DateStr := WORD_TO_STRING(TimeStruct.wDay);
		END_IF
		DateStr := CONCAT(DateStr,'.');
		IF TimeStruct.wMonth < 10 THEN
			DateStr := CONCAT(DateStr,CONCAT('0',WORD_TO_STRING(TimeStruct.wMonth)));
		ELSE
			DateStr := CONCAT(DateStr,WORD_TO_STRING(TimeStruct.wMonth));
		END_IF
		DateStr := CONCAT(DateStr,'.');
		DateStr := CONCAT(DateStr,RIGHT(WORD_TO_STRING(TimeStruct.wYear),2));
	
		(* Time hh.mm.ss.xxms ***************)
		IF TimeStruct.wHour < 10 THEN
			TimeStr := CONCAT('0',WORD_TO_STRING(TimeStruct.wHour));
		ELSE
			TimeStr := WORD_TO_STRING(TimeStruct.wHour);
		END_IF
		TimeStr := CONCAT(TimeStr,':');
		IF TimeStruct.wMinute < 10 THEN
			TimeStr := CONCAT(TimeStr,CONCAT('0',WORD_TO_STRING(TimeStruct.wMinute)));
		ELSE
			TimeStr := CONCAT(TimeStr,WORD_TO_STRING(TimeStruct.wMinute));
		END_IF
		TimeStr := CONCAT(TimeStr,':');
		IF TimeStruct.wSecond < 10 THEN
			TimeStr := CONCAT(TimeStr,CONCAT('0',WORD_TO_STRING(TimeStruct.wSecond)));
		ELSE
			TimeStr := CONCAT(TimeStr,WORD_TO_STRING(TimeStruct.wSecond));
		END_IF
	
		(* TimeStamp Format DE: DD.MM.YY-Stunde:Minute:Sekunde:xxx,*)
		TimeStamp := CONCAT(DateStr,'-');
		TimeStamp := CONCAT(TimeStamp,TimeStr);
		TimeStamp := CONCAT(TimeStamp,':');
		IF TimeStruct.wMilliseconds > 100 THEN
			TimeStamp:=CONCAT(TimeStamp,WORD_TO_STRING(TimeStruct.wMilliseconds));
		ELSIF TimeStruct.wMilliseconds > 10 THEN
			TimeStamp:=CONCAT(CONCAT(TimeStamp,'0'),WORD_TO_STRING(TimeStruct.wMilliseconds));
		ELSE
			TimeStamp:=CONCAT(CONCAT(TimeStamp,'00'),WORD_TO_STRING(TimeStruct.wMilliseconds));
		END_IF
	
		(* Timestamp Format ENG: YYYY-MM-DD-hh:mm:ss.xxx *)
		(* TimeStamp := SYSTEMTIME_TO_STRING(TimeStruct); *)
	
		(* TimeStamp2 FileName YYYY-MM-DD_HHMMSS *)
		IF _sec <> TimeStruct.wSecond THEN
			TimeStamp2 := CONCAT(WORD_TO_STRING(TimeStruct.wYear),'-');
			IF TimeStruct.wMonth < 10 THEN
				TimeStamp2 := CONCAT(TimeStamp2,CONCAT('0',WORD_TO_STRING(TimeStruct.wMonth)));
			ELSE
				TimeStamp2 := CONCAT(TimeStamp2,WORD_TO_STRING(TimeStruct.wMonth));
			END_IF
			TimeStamp2 := CONCAT(TimeStamp2,'-');
			IF TimeStruct.wDay < 10 THEN
				TimeStamp2 := CONCAT(TimeStamp2,CONCAT('0',WORD_TO_STRING(TimeStruct.wDay)));
			ELSE
				TimeStamp2 := CONCAT(TimeStamp2,WORD_TO_STRING(TimeStruct.wDay));
			END_IF
			TimeStamp2 := CONCAT(TimeStamp2,'_');
			IF TimeStruct.wHour < 10 THEN
				TimeStamp2 := CONCAT(TimeStamp2,CONCAT('0',WORD_TO_STRING(TimeStruct.wHour)));
			ELSE
				TimeStamp2 := CONCAT(TimeStamp2,WORD_TO_STRING(TimeStruct.wHour));
			END_IF
			IF TimeStruct.wMinute < 10 THEN
				TimeStamp2 := CONCAT(TimeStamp2,CONCAT('0',WORD_TO_STRING(TimeStruct.wMinute)));
			ELSE
				TimeStamp2 := CONCAT(TimeStamp2,WORD_TO_STRING(TimeStruct.wMinute));
			END_IF
			IF TimeStruct.wSecond < 10 THEN
				TimeStamp2 := CONCAT(TimeStamp2,CONCAT('0',WORD_TO_STRING(TimeStruct.wSecond)));
			ELSE
				TimeStamp2 := CONCAT(TimeStamp2,WORD_TO_STRING(TimeStruct.wSecond));
			END_IF
			_sec := TimeStruct.wSecond;
	
			(* Jahresinformationen *)
			TimeStampDT := SYSTEMTIME_TO_DT(TimeStruct);
			MonthDays	:= F_GetMaxMonthDays(TimeStruct.wYear,TimeStruct.wMonth);
			LeapYear		:= F_YearIsLeapYear(TimeStruct.wYear) ;
			WeekOfYear	:= F_GetWeekOfTheYear(TimeStampDT);
	
		END_IF
	END_IF

(**************************************************************************************************)
END_FUNCTION_BLOCK
ACTION M_Reset:
RetainVarErr := PersistenVarErr := FALSE;
END_ACTION

(* POU 00_Basic/SystemInfo/TaskInfoCtrl, ST *)
FUNCTION_BLOCK TaskInfoCtrl
VAR_INPUT
END_VAR
VAR_OUTPUT
	index						:	INT;
	active					:	BOOL; 		(* Diese Variable zeigt an, ob die Task aktiv ist.*)
	taskName					:	STRING(16);	(* Der Taskname.*)
	firstCycle				:	BOOL;			(* Diese Variable hat im ersten Zyklus der SPS-Task den Wert: TRUE.*)
	cycleTimeExceeded		:	BOOL;			(* In dieser Variablen wird ein 躡erschreiten der eingestellten Taskzykluszeit gemeldet*)
	cycleTime				:	UDINT;		(* Eingestellte Taskzykluszeit in Vielfachen von 100ns*)
	lastExecTime			:	UDINT;		(* Benötigte Zykluszeit für den letzten Zyklus in Vielfachen von 100 ns*)
	MaxExecTime				:	UDINT;		(* Maximale Zykluszeit *)
	priority					:	BYTE;			(* Eingestellte Prioritaet der Task*)
	cycleCount				: 	UDINT;		(* Zykluszaehler*)
END_VAR

VAR
	GETCURTASKINDEX		: GETCURTASKINDEX;
END_VAR
(*********************************************************************************)
	(*	(c) by Hyson Automation																		*)
	(*																											*)
	(*		H Y S O N A U T O M A T I O N   T E C H N O L O G Y        *)
	(*																											*)
	(*		Rd.Keyuan16	Shenzhen	China	phone:	+86-755-28376157	www.hyson-au.cn	*)
   (*																											*)
   (*		Content					: Hyson Program Framework													*)
	(*																											*)
	(*		Version					:	V2.10																	*)
	(*		Stand					:	04.2020																*)
 	(*		Autor					:	ShenQiang															*)
	(*																											*)
	(*********************************************************************************)

(* Get Current Task Index ************************************************************************)
	GETCURTASKINDEX(index => index);

	(* Retein/Persisten Data Err *)
	active := SystemTaskInfoArr[index].active;
	taskName := SystemTaskInfoArr[index].taskName;
	firstCycle := SystemTaskInfoArr[index].firstCycle;
	cycleTimeExceeded := SystemTaskInfoArr[index].cycleTimeExceeded;
	cycleTime := SystemTaskInfoArr[index].cycleTime;
	lastExecTime := SystemTaskInfoArr[index].lastExecTime;
	MaxExecTime	:= MAX(lastExecTime,MaxExecTime);
	priority := SystemTaskInfoArr[index].priority;
	firstCycle := SystemTaskInfoArr[index].firstCycle;
	cycleCount := SystemTaskInfoArr[index].cycleCount;

(**************************************************************************************************)
END_FUNCTION_BLOCK
